        IF rtb_IP_boBMS_HV_REL_ON_BB3 THEN 
            Count_k := REAL_TO_LREAL(rtb_Add_m);
        ELSE 
            Count_k := 65535.0;
        END_IF;

        (* End of Switch: '<S128>/Switch2' *)
        (* End of Outputs for SubSystem: '<S676>/BatteryPackSignals' *)
        

        (* Switch: '<S128>/Switch3' incorporates:
         *  Constant: '<S128>/Constant5'
         *  Constant: '<S129>/Constant'
         *  Constant: '<S130>/Constant'
         *  Constant: '<S131>/Constant'
         *  Constant: '<S132>/Constant'
         *  Constant: '<S133>/Constant'
         *  Constant: '<S134>/Constant'
         *  Constant: '<S135>/Constant'
         *  Constant: '<S136>/Constant'
         *  Constant: '<S137>/Constant'
         *  Logic: '<S128>/AND'
         *  Logic: '<S128>/AND1'
         *  Logic: '<S128>/AND2'
         *  RelationalOperator: '<S129>/Compare'
         *  RelationalOperator: '<S130>/Compare'
         *  RelationalOperator: '<S131>/Compare'
         *  RelationalOperator: '<S132>/Compare'
         *  RelationalOperator: '<S133>/Compare'
         *  RelationalOperator: '<S134>/Compare'
         *  RelationalOperator: '<S135>/Compare'
         *  RelationalOperator: '<S136>/Compare'
         *  RelationalOperator: '<S137>/Compare'
         *  Switch: '<S128>/Switch4'
         *  Switch: '<S128>/Switch5' *)

        IF ((rtb_Uk1 >= 15.0) AND (rtb_UnitDelay2 >= 15.0)) AND (Count_k >= 15.0) THEN 
            rtb_Switch3 := CurrentReductionConstant_Lvl3;
        ELSIF ((rtb_Uk1 >= 10.0) AND (rtb_UnitDelay2 >= 10.0)) AND (Count_k >= 10.0) THEN 
            (* Switch: '<S128>/Switch4' incorporates:
             *  Constant: '<S128>/Constant3' *)
            rtb_Switch3 := CurrentReductionConstant_Lvl2;
        ELSIF ((rtb_Uk1 >= 5.0) AND (rtb_UnitDelay2 >= 5.0)) AND (Count_k >= 5.0) THEN 
            (* Switch: '<S128>/Switch5' incorporates:
             *  Constant: '<S128>/Constant4'
             *  Switch: '<S128>/Switch4' *)
            rtb_Switch3 := CurrentReductionConstant_Lvl1;
        ELSE 
            (* Switch: '<S128>/Switch5' incorporates:
             *  Constant: '<S128>/Constant6'
             *  Switch: '<S128>/Switch4' *)
            rtb_Switch3 := CurrentReductionConstant_Lvl0;
        END_IF;

        (* End of Switch: '<S128>/Switch3' *)
        

        (* Outputs for Atomic SubSystem: '<S676>/BatteryPackSignals' *)
        (* Product: '<S110>/Product2' incorporates:
         *  Constant: '<S110>/Constant'
         *  Constant: '<S110>/Constant5'
         *  Constant: '<S110>/Constant6'
         *  Constant: '<S126>/Constant'
         *  Logic: '<S110>/AND'
         *  MinMax: '<S110>/Min'
         *  RelationalOperator: '<S126>/Compare'
         *  RelationalOperator: '<S127>/Compare'
         *  SignalConversion: '<S682>/BusConversion_InsertedFor_IT_BatterySignal_Databus_at_inport_0'
         *  Sum: '<S110>/Add' *)

        IF rtb_NOT_m5 THEN 
            b_temp3 := MIN(rtb_Switch5_bs, rtb_Add_ci);
            temp3 := MIN(b_temp3, rtb_Divide_h) * USINT_TO_REAL(rtb_ExtractDesiredBits_bk_tmp);
        ELSE 
            temp3 := 0.0;
        END_IF;

        i0_BattChargeFcn(ssMethodType := SS_OUTPUT, MaxChargeCurr_fb := rtb_UnitDelay, MaxChargeCurrentBatt := temp3, ChargeStopPressed := rtb_IT_boChargeStop_Button, HV_ON_Batt1 := rtb_IP_boBMS_HV_REL_ON_BB1, HV_ON_Batt2 := rtb_IP_boBMS_HV_REL_ON_BB2, HV_ON_Batt3 := rtb_IP_boBMS_HV_REL_ON_BB3, Ibatt1 := rtb_Add_ki5, Ibatt2 := rtb_Add_ir, Ibatt3 := rtb_Add_m, Fcn_available := (UnexpectedBattChargingFcn_Available AND (rtb_ExtractDesiredBits_bk_tmp > 1)) AND ( NOT rtb_FL_boKL15_Disable), CurrentReductionConstant := rtb_Switch3, CurrentLB_f := CurrentLB, CurrentUB_c := CurrentUB);
        FL_sST_MaxChargeCurrent := i0_BattChargeFcn.FL_sST_MaxChargeCurrent;
        REQ_HV_Open_Batt2 := i0_BattChargeFcn.REQ_HV_Open_Batt2;
        REQ_HV_Open_Batt3 := i0_BattChargeFcn.REQ_HV_Open_Batt3;
        REQ_HV_Open_Batt1 := i0_BattChargeFcn.REQ_HV_Open_Batt1;
        BatteryReadyToShutDown := i0_BattChargeFcn.BatteryReadyToShutDown;
        (* End of Outputs for SubSystem: '<S676>/BatteryPackSignals' *)
        

        (* Switch: '<S116>/Switch' incorporates:
         *  Abs: '<S116>/Abs'
         *  Abs: '<S116>/Abs1'
         *  Abs: '<S116>/Abs2'
         *  Constant: '<S116>/Constant'
         *  Constant: '<S187>/Constant'
         *  Constant: '<S188>/Constant'
         *  Constant: '<S189>/Constant'
         *  Logic: '<S116>/AND'
         *  Logic: '<S116>/AND1'
         *  Logic: '<S116>/AND2'
         *  RelationalOperator: '<S187>/Compare'
         *  RelationalOperator: '<S188>/Compare'
         *  RelationalOperator: '<S189>/Compare'
         *  SignalConversion: '<S682>/BusConversion_InsertedFor_IT_BatterySignal_Databus_at_inport_0' *)

        IF UnexpectedBattChargingFcn_Available THEN 
            (* Outputs for Atomic SubSystem: '<S676>/BatteryPackSignals' *)
            rtb_IT_boChargeStop_Button := ((((ABS(rtb_Add_ki5) <= 1.0) AND (ABS(rtb_Add_ir) <= 1.0)) AND (ABS(rtb_Add_m) <= 1.0)) AND rtb_IT_boUDC_SafeToShutdown) OR (rtb_IT_boUDC_SafeToShutdown AND BatteryReadyToShutDown);
            (* End of Outputs for SubSystem: '<S676>/BatteryPackSignals' *)
        ELSE 
            rtb_IT_boChargeStop_Button := rtb_IT_boUDC_SafeToShutdown;
        END_IF;

        (* End of Switch: '<S116>/Switch' *)
        

        (* SignalConversion: '<S13>/TmpSignal ConversionAtChart_REQ_MAIN_MINUSInport4' *)
        i0_Chart_REQ_MAIN_MINUS(ssMethodType := SS_OUTPUT, In := rtb_Out_bl, CM_SafeToSD := rtb_IT_boChargeStop_Button, KL15_CM_disable := rtb_FL_boKL15_Disable, System_ESD := rtb_UnitDelay1_d, System_SD := rtb_UnitDelay1_d, b_Reset := rtb_FL_boSS_BDU_Reset);
        REQ_MainHV_ON_MINUS_g := i0_Chart_REQ_MAIN_MINUS.REQ_MainHV_ON_MINUS;
        (* Logic: '<S21>/AND3' incorporates:
         *  Constant: '<S13>/Constant'
         *  RelationalOperator: '<S29>/FixPt Relational Operator'
         *  UnitDelay: '<S29>/Delay Input1'
         *
         * Block description for '<S29>/Delay Input1':
         *  
         *  Store in Global RAM *)
        rtb_IT_boChargeStop_Button := (DelayInput1_DSTATE > 0.0) AND rtb_FL_boKL15_Disable;
        (* MinMax: '<S120>/Min' *)
        i0_Chart_WeldingDetection(ssMethodType := SS_OUTPUT, LoadVtg := DINT_TO_REAL(rtb_Add_kr), SystemVtg := maxV, In := rtb_IT_boChargeStop_Button);
        MainHV_Minus_Welded := i0_Chart_WeldingDetection.MainHV_Minus_Welded;
        MainHV_Plus_Welded := i0_Chart_WeldingDetection.MainHV_Plus_Welded;
        REQ_MainHV_ON_MINUS := i0_Chart_WeldingDetection.REQ_MainHV_ON_MINUS;
        REQ_MainHV_ON_PLUS := i0_Chart_WeldingDetection.REQ_MainHV_ON_PLUS;
        WeldingDetection_Status := i0_Chart_WeldingDetection.WeldingDetection_Status;
        (* UnitDelay: '<S21>/Unit Delay' *)
        rtb_System_SD_ErrorCode := UnitDelay_DSTATE_i;
        (* Chart: '<S21>/Chart4' *)
        (* Gateway: ChiefMaster/Flow Logic/BDU Control/BDUSystem/Subsystem1/Chart4 *)
        (* During: ChiefMaster/Flow Logic/BDU Control/BDUSystem/Subsystem1/Chart4 *)
        temp1 := FALSE;
        temp2 := FALSE;

        IF is_active_c46_ChiefMaster = 0 THEN 
            (* Entry: ChiefMaster/Flow Logic/BDU Control/BDUSystem/Subsystem1/Chart4 *)
            is_active_c46_ChiefMaster := 1;
            (* Entry Internal: ChiefMaster/Flow Logic/BDU Control/BDUSystem/Subsystem1/Chart4 *)
            (* Transition: '<S28>:2' *)
            is_c46_ChiefMaster := ChiefMaster_IN_Default_e2;
            (* Entry 'Default': '<S28>:1' *)
            (* '<S28>:1:2' Out = false *)
            rtb_Out_k := FALSE;
            temp1 := TRUE;
        ELSE 

            CASE is_c46_ChiefMaster OF
                ChiefMaster_IN_Default_e2: 
                    (* During 'Default': '<S28>:1' *)
                    (* '<S28>:5:1' sf_internal_predicateOutput = In == true; *)

                    IF rtb_IT_boChargeStop_Button THEN 
                        (* Transition: '<S28>:5' *)
                        is_c46_ChiefMaster := ChiefMaster_IN_Default1;
                        (* Entry 'Default1': '<S28>:4' *)
                        (* '<S28>:4:2' Out = true *)
                        rtb_Out_k := TRUE;
                        temp2 := TRUE;
                    ELSE 
                        (* '<S28>:1:2' Out = false *)
                        rtb_Out_k := FALSE;
                        temp1 := TRUE;
                    END_IF;

                ELSE
                    (* During 'Default1': '<S28>:4' *)
                    (* '<S28>:9:1' sf_internal_predicateOutput = WeldingDetection_Status == 1 ||... *)
                    (* '<S28>:9:2' WeldingDetection_Status == 2; *)

                    IF (rtb_System_SD_ErrorCode = 1) OR (rtb_System_SD_ErrorCode = 2) THEN 
                        (* Transition: '<S28>:9' *)
                        is_c46_ChiefMaster := ChiefMaster_IN_Default_e2;
                        (* Entry 'Default': '<S28>:1' *)
                        (* '<S28>:1:2' Out = false *)
                        rtb_Out_k := FALSE;
                        temp1 := TRUE;
                    ELSE 
                        (* '<S28>:4:2' Out = true *)
                        rtb_Out_k := TRUE;
                        temp2 := TRUE;
                    END_IF;

            END_CASE;

        END_IF;


        IF temp2 THEN 
            (* Switch: '<S13>/Switch' *)
            DO_REQ_MainHV_ON_MINUS := REQ_MainHV_ON_MINUS;
            (* Switch: '<S13>/Switch1' *)
            DO_REQ_MainHV_ON_PLUS := REQ_MainHV_ON_PLUS;
        END_IF;


        IF temp1 THEN 
            (* Switch: '<S13>/Switch' *)
            DO_REQ_MainHV_ON_MINUS := REQ_MainHV_ON_MINUS_g;
            (* Switch: '<S13>/Switch1' incorporates:
             *  Constant: '<S18>/Constant'
             *  Logic: '<S13>/AND5'
             *  RelationalOperator: '<S18>/Compare'
             *  RelationalOperator: '<S19>/Compare' *)
            DO_REQ_MainHV_ON_PLUS := ((Precharge_Satus = 1.0) AND rtb_IT_boHW_MainHV_Minus_FB) AND REQ_MainHV_ON_MINUS_g;
        END_IF;

        (* End of Chart: '<S21>/Chart4' *)
        

        (* Chart: '<S20>/Chart_Main_Minus_Status' incorporates:
         *  Constant: '<S20>/Constant2' *)
        (* Gateway: ChiefMaster/Flow Logic/BDU Control/BDUSystem/Subsystem/Chart_Main_Minus_Status *)
        (* During: ChiefMaster/Flow Logic/BDU Control/BDUSystem/Subsystem/Chart_Main_Minus_Status *)

        IF is_active_c40_ChiefMaster = 0 THEN 
            (* Entry: ChiefMaster/Flow Logic/BDU Control/BDUSystem/Subsystem/Chart_Main_Minus_Status *)
            is_active_c40_ChiefMaster := 1;
            (* Entry Internal: ChiefMaster/Flow Logic/BDU Control/BDUSystem/Subsystem/Chart_Main_Minus_Status *)
            (* Transition: '<S26>:2' *)
            is_c40_ChiefMaster := ChiefMaster_IN_Default_e2;
            (* Entry 'Default': '<S26>:1' *)
            (* '<S26>:1:2' MainHV_Minus_Status = 0 *)
            MainHV_Minus_Status := 0.0;
        ELSE 

            CASE is_c40_ChiefMaster OF
                ChiefMaster_IN_Default_e2: 
                    (* During 'Default': '<S26>:1' *)
                    (* '<S26>:10:1' sf_internal_predicateOutput = REQ_MainHV_ON_MINUS == false &&... *)
                    (* '<S26>:10:2' CMShutdown == false; *)

                    IF ( NOT DO_REQ_MainHV_ON_MINUS) AND ( NOT rtb_FL_boCMSleep) THEN 
                        (* Transition: '<S26>:10' *)
                        is_c40_ChiefMaster := ChiefMaster_IN_hold_a;
                        temporalCounter_i1_k(timerAction := 1, maxTime := 0);
                        (* Entry 'hold': '<S26>:9' *)
                        (* '<S26>:9:2' MainHV_Minus_Status = 0 *)
                        MainHV_Minus_Status := 0.0;
                    ELSE 
                        (* '<S26>:1:2' MainHV_Minus_Status = 0 *)
                        MainHV_Minus_Status := 0.0;
                    END_IF;

                ChiefMaster_IN_Error_p: 
                    (* During 'Error': '<S26>:16' *)
                    (* '<S26>:51:1' sf_internal_predicateOutput = CMShutdown == true; *)

                    IF rtb_FL_boCMSleep THEN 
                        (* Transition: '<S26>:51' *)
                        is_c40_ChiefMaster := ChiefMaster_IN_Default_e2;
                        (* Entry 'Default': '<S26>:1' *)
                        (* '<S26>:1:2' MainHV_Minus_Status = 0 *)
                        MainHV_Minus_Status := 0.0;
                    ELSE 
                        (* '<S26>:16:2' MainHV_Minus_Status = 3 *)
                        MainHV_Minus_Status := 3.0;
                    END_IF;

                ChiefMaster_IN_closed: 
                    (* During 'closed': '<S26>:38' *)
                    (* '<S26>:44:1' sf_internal_predicateOutput = REQ_MainHV_ON_MINUS == false; *)

                    IF  NOT DO_REQ_MainHV_ON_MINUS THEN 
                        (* Transition: '<S26>:44' *)
                        (* Transition: '<S26>:45' *)
                        (* Transition: '<S26>:49' *)
                        is_c40_ChiefMaster := ChiefMaster_IN_hold_a;
                        temporalCounter_i1_k(timerAction := 1, maxTime := 0);
                        (* Entry 'hold': '<S26>:9' *)
                        (* '<S26>:9:2' MainHV_Minus_Status = 0 *)
                        MainHV_Minus_Status := 0.0;
                    ELSE 
                        (* '<S26>:41:1' sf_internal_predicateOutput = MainHV_ON_Minus_FB == false; *)

                        IF  NOT rtb_IT_boHW_MainHV_Minus_FB THEN 
                            (* Transition: '<S26>:41' *)
                            (* Transition: '<S26>:42' *)
                            (* Transition: '<S26>:29' *)
                            (* Transition: '<S26>:27' *)
                            is_c40_ChiefMaster := ChiefMaster_IN_Error_p;
                            (* Entry 'Error': '<S26>:16' *)
                            (* '<S26>:16:2' MainHV_Minus_Status = 3 *)
                            MainHV_Minus_Status := 3.0;
                        ELSE 
                            (* '<S26>:38:2' MainHV_Minus_Status = 2 *)
                            MainHV_Minus_Status := 2.0;
                        END_IF;

                    END_IF;

                ChiefMaster_IN_hold_a: 
                    (* During 'hold': '<S26>:9' *)
                    (* '<S26>:5:1' sf_internal_predicateOutput = MainHV_ON_Minus_FB == false; *)

                    IF  NOT rtb_IT_boHW_MainHV_Minus_FB THEN 
                        (* Transition: '<S26>:5' *)
                        is_c40_ChiefMaster := ChiefMaster_IN_open;
                        (* Entry 'open': '<S26>:4' *)
                        (* '<S26>:4:2' MainHV_Minus_Status = 1 *)
                        MainHV_Minus_Status := 1.0;
                    ELSE 
                        (* '<S26>:17:1' sf_internal_predicateOutput = after(DelayTime_s,sec); *)
                        temporalCounter_i1_k(timerAction := 2, maxTime := TRUNC(REAL_TO_LREAL(MainHV_StatusDelay) * 1000.0));

                        IF temporalCounter_i1_k.done THEN 
                            (* Transition: '<S26>:17' *)
                            is_c40_ChiefMaster := ChiefMaster_IN_Error_p;
                            (* Entry 'Error': '<S26>:16' *)
                            (* '<S26>:16:2' MainHV_Minus_Status = 3 *)
                            MainHV_Minus_Status := 3.0;
                        ELSE 
                            (* '<S26>:9:2' MainHV_Minus_Status = 0 *)
                            MainHV_Minus_Status := 0.0;
                        END_IF;

                    END_IF;

                ChiefMaster_IN_hold1: 
                    (* During 'hold1': '<S26>:23' *)
                    (* '<S26>:39:1' sf_internal_predicateOutput = MainHV_ON_Minus_FB == true; *)

                    IF rtb_IT_boHW_MainHV_Minus_FB THEN 
                        (* Transition: '<S26>:39' *)
                        is_c40_ChiefMaster := ChiefMaster_IN_closed;
                        (* Entry 'closed': '<S26>:38' *)
                        (* '<S26>:38:2' MainHV_Minus_Status = 2 *)
                        MainHV_Minus_Status := 2.0;
                    ELSE 
                        (* '<S26>:26:1' sf_internal_predicateOutput = after(DelayTime_s,sec); *)
                        temporalCounter_i1_k(timerAction := 2, maxTime := TRUNC(REAL_TO_LREAL(MainHV_StatusDelay) * 1000.0));

                        IF temporalCounter_i1_k.done THEN 
                            (* Transition: '<S26>:26' *)
                            (* Transition: '<S26>:29' *)
                            (* Transition: '<S26>:27' *)
                            is_c40_ChiefMaster := ChiefMaster_IN_Error_p;
                            (* Entry 'Error': '<S26>:16' *)
                            (* '<S26>:16:2' MainHV_Minus_Status = 3 *)
                            MainHV_Minus_Status := 3.0;
                        ELSE 
                            (* '<S26>:23:2' MainHV_Minus_Status = 1 *)
                            MainHV_Minus_Status := 1.0;
                        END_IF;

                    END_IF;

                ELSE
                    (* During 'open': '<S26>:4' *)
                    (* '<S26>:11:1' sf_internal_predicateOutput = REQ_MainHV_ON_MINUS == true; *)

                    IF DO_REQ_MainHV_ON_MINUS THEN 
                        (* Transition: '<S26>:11' *)
                        is_c40_ChiefMaster := ChiefMaster_IN_hold1;
                        temporalCounter_i1_k(timerAction := 1, maxTime := 0);
                        (* Entry 'hold1': '<S26>:23' *)
                        (* '<S26>:23:2' MainHV_Minus_Status = 1 *)
                        MainHV_Minus_Status := 1.0;
                    ELSE 
                        (* '<S26>:19:1' sf_internal_predicateOutput = MainHV_ON_Minus_FB == true; *)

                        IF rtb_IT_boHW_MainHV_Minus_FB THEN 
                            (* Transition: '<S26>:19' *)
                            (* Transition: '<S26>:27' *)
                            is_c40_ChiefMaster := ChiefMaster_IN_Error_p;
                            (* Entry 'Error': '<S26>:16' *)
                            (* '<S26>:16:2' MainHV_Minus_Status = 3 *)
                            MainHV_Minus_Status := 3.0;
                        ELSE 
                            (* '<S26>:4:2' MainHV_Minus_Status = 1 *)
                            MainHV_Minus_Status := 1.0;
                        END_IF;

                    END_IF;

            END_CASE;

        END_IF;

        (* End of Chart: '<S20>/Chart_Main_Minus_Status' *)
        (* End of Outputs for SubSystem: '<Root>/ChiefMaster' *)
        

        (* Constant: '<S390>/Constant4' incorporates:
         *  Constant: '<S390>/Constant'
         *  Constant: '<S390>/Constant1'
         *  Constant: '<S390>/Constant2'
         *  Constant: '<S390>/Constant3' *)
        i2_Chart_Hysteresis_LowActive(ssMethodType := SS_OUTPUT, sSignal := AI_MainHV_Plus_FB, boInitial_Value := FALSE, boValue_Activated := TRUE, boValue_Deactivated := FALSE, sLB := 5000.0, b_sUB := 10000.0);
        boOutput_o := i2_Chart_Hysteresis_LowActive.boOutput;
        (* Outputs for Atomic SubSystem: '<Root>/ChiefMaster' *)
        (* SignalConversion: '<S677>/Signal Copy4' *)
        rtb_IT_boHW_MainHV_Plus_FB := boOutput_o;
        (* Chart: '<S20>/Chart_Main_Plus_Status' incorporates:
         *  Constant: '<S20>/Constant2'
         *  SignalConversion: '<S677>/Signal Copy4' *)
        (* Gateway: ChiefMaster/Flow Logic/BDU Control/BDUSystem/Subsystem/Chart_Main_Plus_Status *)
        (* During: ChiefMaster/Flow Logic/BDU Control/BDUSystem/Subsystem/Chart_Main_Plus_Status *)

        IF is_active_c41_ChiefMaster = 0 THEN 
            (* Entry: ChiefMaster/Flow Logic/BDU Control/BDUSystem/Subsystem/Chart_Main_Plus_Status *)
            is_active_c41_ChiefMaster := 1;
            (* Entry Internal: ChiefMaster/Flow Logic/BDU Control/BDUSystem/Subsystem/Chart_Main_Plus_Status *)
            (* Transition: '<S27>:2' *)
            is_c41_ChiefMaster := ChiefMaster_IN_Default_e2;
            (* Entry 'Default': '<S27>:1' *)
            (* '<S27>:1:2' MainHV_Plus_Status = 0 *)
            MainHV_Plus_Status := 0.0;
        ELSE 

            CASE is_c41_ChiefMaster OF
                ChiefMaster_IN_Default_e2: 
                    (* During 'Default': '<S27>:1' *)
                    (* '<S27>:10:1' sf_internal_predicateOutput = REQ_MainHV_ON_PLUS == false &&... *)
                    (* '<S27>:10:2' CMShutdown == false; *)

                    IF ( NOT DO_REQ_MainHV_ON_PLUS) AND ( NOT rtb_FL_boCMSleep) THEN 
                        (* Transition: '<S27>:10' *)
                        is_c41_ChiefMaster := ChiefMaster_IN_hold_a;
                        temporalCounter_i1_he(timerAction := 1, maxTime := 0);
                        (* Entry 'hold': '<S27>:9' *)
                        (* '<S27>:9:2' MainHV_Plus_Status = 0 *)
                        MainHV_Plus_Status := 0.0;
                    ELSE 
                        (* '<S27>:1:2' MainHV_Plus_Status = 0 *)
                        MainHV_Plus_Status := 0.0;
                    END_IF;

                ChiefMaster_IN_Error_p: 
                    (* During 'Error': '<S27>:16' *)
                    (* '<S27>:50:1' sf_internal_predicateOutput = CMShutdown == true; *)

                    IF rtb_FL_boCMSleep THEN 
                        (* Transition: '<S27>:50' *)
                        is_c41_ChiefMaster := ChiefMaster_IN_Default_e2;
                        (* Entry 'Default': '<S27>:1' *)
                        (* '<S27>:1:2' MainHV_Plus_Status = 0 *)
                        MainHV_Plus_Status := 0.0;
                    ELSE 
                        (* '<S27>:16:2' MainHV_Plus_Status = 3 *)
                        MainHV_Plus_Status := 3.0;
                    END_IF;

                ChiefMaster_IN_closed: 
                    (* During 'closed': '<S27>:38' *)
                    (* '<S27>:44:1' sf_internal_predicateOutput = REQ_MainHV_ON_PLUS == false; *)

                    IF  NOT DO_REQ_MainHV_ON_PLUS THEN 
                        (* Transition: '<S27>:44' *)
                        (* Transition: '<S27>:45' *)
                        (* Transition: '<S27>:49' *)
                        is_c41_ChiefMaster := ChiefMaster_IN_hold_a;
                        temporalCounter_i1_he(timerAction := 1, maxTime := 0);
                        (* Entry 'hold': '<S27>:9' *)
                        (* '<S27>:9:2' MainHV_Plus_Status = 0 *)
                        MainHV_Plus_Status := 0.0;
                    ELSE 
                        (* '<S27>:54:1' sf_internal_predicateOutput = MainHV_ON_Plus_FB == false; *)

                        IF  NOT boOutput_o THEN 
                            (* Transition: '<S27>:54' *)
                            (* Transition: '<S27>:42' *)
                            (* Transition: '<S27>:67' *)
                            (* Transition: '<S27>:59' *)
                            is_c41_ChiefMaster := ChiefMaster_IN_Error_p;
                            (* Entry 'Error': '<S27>:16' *)
                            (* '<S27>:16:2' MainHV_Plus_Status = 3 *)
                            MainHV_Plus_Status := 3.0;
                        ELSE 
                            (* '<S27>:38:2' MainHV_Plus_Status = 2 *)
                            MainHV_Plus_Status := 2.0;
                        END_IF;

                    END_IF;

                ChiefMaster_IN_hold_a: 
                    (* During 'hold': '<S27>:9' *)
                    (* '<S27>:5:1' sf_internal_predicateOutput = MainHV_ON_Plus_FB == false; *)

                    IF  NOT boOutput_o THEN 
                        (* Transition: '<S27>:5' *)
                        is_c41_ChiefMaster := ChiefMaster_IN_open;
                        (* Entry 'open': '<S27>:4' *)
                        (* '<S27>:4:2' MainHV_Plus_Status = 1 *)
                        MainHV_Plus_Status := 1.0;
                    ELSE 
                        (* '<S27>:17:1' sf_internal_predicateOutput = after(DelayTime_s,sec); *)
                        temporalCounter_i1_he(timerAction := 2, maxTime := TRUNC(REAL_TO_LREAL(MainHV_StatusDelay) * 1000.0));

                        IF temporalCounter_i1_he.done THEN 
                            (* Transition: '<S27>:17' *)
                            is_c41_ChiefMaster := ChiefMaster_IN_Error_p;
                            (* Entry 'Error': '<S27>:16' *)
                            (* '<S27>:16:2' MainHV_Plus_Status = 3 *)
                            MainHV_Plus_Status := 3.0;
                        ELSE 
                            (* '<S27>:9:2' MainHV_Plus_Status = 0 *)
                            MainHV_Plus_Status := 0.0;
                        END_IF;

                    END_IF;

                ChiefMaster_IN_hold1: 
                    (* During 'hold1': '<S27>:23' *)
                    (* '<S27>:39:1' sf_internal_predicateOutput = MainHV_ON_Plus_FB == true; *)

                    IF boOutput_o THEN 
                        (* Transition: '<S27>:39' *)
                        is_c41_ChiefMaster := ChiefMaster_IN_closed;
                        (* Entry 'closed': '<S27>:38' *)
                        (* '<S27>:38:2' MainHV_Plus_Status = 2 *)
                        MainHV_Plus_Status := 2.0;
                    ELSE 
                        (* '<S27>:26:1' sf_internal_predicateOutput = after(DelayTime_s,sec); *)
                        temporalCounter_i1_he(timerAction := 2, maxTime := TRUNC(REAL_TO_LREAL(MainHV_StatusDelay) * 1000.0));

                        IF temporalCounter_i1_he.done THEN 
                            (* Transition: '<S27>:26' *)
                            (* Transition: '<S27>:67' *)
                            (* Transition: '<S27>:59' *)
                            is_c41_ChiefMaster := ChiefMaster_IN_Error_p;
                            (* Entry 'Error': '<S27>:16' *)
                            (* '<S27>:16:2' MainHV_Plus_Status = 3 *)
                            MainHV_Plus_Status := 3.0;
                        ELSE 
                            (* '<S27>:23:2' MainHV_Plus_Status = 1 *)
                            MainHV_Plus_Status := 1.0;
                        END_IF;

                    END_IF;

                ELSE
                    (* During 'open': '<S27>:4' *)
                    (* '<S27>:11:1' sf_internal_predicateOutput = REQ_MainHV_ON_PLUS == true; *)

                    IF DO_REQ_MainHV_ON_PLUS THEN 
                        (* Transition: '<S27>:11' *)
                        is_c41_ChiefMaster := ChiefMaster_IN_hold1;
                        temporalCounter_i1_he(timerAction := 1, maxTime := 0);
                        (* Entry 'hold1': '<S27>:23' *)
                        (* '<S27>:23:2' MainHV_Plus_Status = 1 *)
                        MainHV_Plus_Status := 1.0;
                    ELSE 
                        (* '<S27>:58:1' sf_internal_predicateOutput = MainHV_ON_Plus_FB == true; *)

                        IF boOutput_o THEN 
                            (* Transition: '<S27>:58' *)
                            (* Transition: '<S27>:59' *)
                            is_c41_ChiefMaster := ChiefMaster_IN_Error_p;
                            (* Entry 'Error': '<S27>:16' *)
                            (* '<S27>:16:2' MainHV_Plus_Status = 3 *)
                            MainHV_Plus_Status := 3.0;
                        ELSE 
                            (* '<S27>:4:2' MainHV_Plus_Status = 1 *)
                            MainHV_Plus_Status := 1.0;
                        END_IF;

                    END_IF;

            END_CASE;

        END_IF;

        (* End of Chart: '<S20>/Chart_Main_Plus_Status' *)
        (* End of Outputs for SubSystem: '<Root>/ChiefMaster' *)
        

        (* Constant: '<S389>/Constant4' incorporates:
         *  Constant: '<S389>/Constant'
         *  Constant: '<S389>/Constant1'
         *  Constant: '<S389>/Constant2'
         *  Constant: '<S389>/Constant3' *)
        i1_Chart_Hysteresis_LowActive(ssMethodType := SS_OUTPUT, sSignal := AI_DCHV_Minus_FB, boInitial_Value := FALSE, boValue_Activated := TRUE, boValue_Deactivated := FALSE, sLB := 5000.0, b_sUB := 10000.0);
        boOutput_a := i1_Chart_Hysteresis_LowActive.boOutput;
        (* Outputs for Atomic SubSystem: '<Root>/ChiefMaster' *)
        (* SignalConversion: '<S677>/Signal Copy13' *)
        rtb_IT_boHW_DCHV_Minus_FB := boOutput_a;
        (* Chart: '<S23>/Chart_DCMinus_Status' incorporates:
         *  Constant: '<S23>/Constant2'
         *  SignalConversion: '<S677>/Signal Copy13' *)
        (* Gateway: ChiefMaster/Flow Logic/BDU Control/BDUSystem/Subsystem3/Chart_DCMinus_Status *)
        (* During: ChiefMaster/Flow Logic/BDU Control/BDUSystem/Subsystem3/Chart_DCMinus_Status *)

        IF is_active_c53_ChiefMaster = 0 THEN 
            (* Entry: ChiefMaster/Flow Logic/BDU Control/BDUSystem/Subsystem3/Chart_DCMinus_Status *)
            is_active_c53_ChiefMaster := 1;
            (* Entry Internal: ChiefMaster/Flow Logic/BDU Control/BDUSystem/Subsystem3/Chart_DCMinus_Status *)
            (* Transition: '<S31>:2' *)
            is_c53_ChiefMaster := ChiefMaster_IN_Default_e2;
            (* Entry 'Default': '<S31>:1' *)
            (* '<S31>:1:2' HV_Minus_Status = 0 *)
            rtb_Uk1 := 0.0;
        ELSE 

            CASE is_c53_ChiefMaster OF
                ChiefMaster_IN_Default_e2: 
                    (* During 'Default': '<S31>:1' *)
                    (* '<S31>:10:1' sf_internal_predicateOutput = REQ_HV_ON_MINUS == false &&... *)
                    (* '<S31>:10:2' CMSleep == false; *)

                    IF ( NOT DO_REQ_DC_ON_PLUS) AND ( NOT rtb_FL_boCMSleep) THEN 
                        (* Transition: '<S31>:10' *)
                        is_c53_ChiefMaster := ChiefMaster_IN_hold_a;
                        temporalCounter_i1_n(timerAction := 1, maxTime := 0);
                        (* Entry 'hold': '<S31>:9' *)
                        (* '<S31>:9:2' HV_Minus_Status = 0 *)
                        rtb_Uk1 := 0.0;
                    ELSE 
                        (* '<S31>:1:2' HV_Minus_Status = 0 *)
                        rtb_Uk1 := 0.0;
                    END_IF;

                ChiefMaster_IN_Error_p: 
                    (* During 'Error': '<S31>:16' *)
                    (* '<S31>:51:1' sf_internal_predicateOutput = CMSleep == true; *)

                    IF rtb_FL_boCMSleep THEN 
                        (* Transition: '<S31>:51' *)
                        is_c53_ChiefMaster := ChiefMaster_IN_Default_e2;
                        (* Entry 'Default': '<S31>:1' *)
                        (* '<S31>:1:2' HV_Minus_Status = 0 *)
                        rtb_Uk1 := 0.0;
                    ELSE 
                        (* '<S31>:16:2' HV_Minus_Status = 3 *)
                        rtb_Uk1 := 3.0;
                    END_IF;

                ChiefMaster_IN_closed: 
                    (* During 'closed': '<S31>:38' *)
                    (* '<S31>:44:1' sf_internal_predicateOutput = REQ_HV_ON_MINUS == false; *)

                    IF  NOT DO_REQ_DC_ON_PLUS THEN 
                        (* Transition: '<S31>:44' *)
                        (* Transition: '<S31>:45' *)
                        (* Transition: '<S31>:49' *)
                        is_c53_ChiefMaster := ChiefMaster_IN_hold_a;
                        temporalCounter_i1_n(timerAction := 1, maxTime := 0);
                        (* Entry 'hold': '<S31>:9' *)
                        (* '<S31>:9:2' HV_Minus_Status = 0 *)
                        rtb_Uk1 := 0.0;
                    ELSE 
                        (* '<S31>:41:1' sf_internal_predicateOutput = HV_ON_Minus_FB == false; *)

                        IF  NOT boOutput_a THEN 
                            (* Transition: '<S31>:41' *)
                            (* Transition: '<S31>:42' *)
                            (* Transition: '<S31>:29' *)
                            (* Transition: '<S31>:27' *)
                            is_c53_ChiefMaster := ChiefMaster_IN_Error_p;
                            (* Entry 'Error': '<S31>:16' *)
                            (* '<S31>:16:2' HV_Minus_Status = 3 *)
                            rtb_Uk1 := 3.0;
                        ELSE 
                            (* '<S31>:38:2' HV_Minus_Status = 2 *)
                            rtb_Uk1 := 2.0;
                        END_IF;

                    END_IF;

                ChiefMaster_IN_hold_a: 
                    (* During 'hold': '<S31>:9' *)
                    (* '<S31>:5:1' sf_internal_predicateOutput = HV_ON_Minus_FB == false; *)

                    IF  NOT boOutput_a THEN 
                        (* Transition: '<S31>:5' *)
                        is_c53_ChiefMaster := ChiefMaster_IN_open;
                        (* Entry 'open': '<S31>:4' *)
                        (* '<S31>:4:2' HV_Minus_Status = 1 *)
                        rtb_Uk1 := 1.0;
                    ELSE 
                        (* '<S31>:17:1' sf_internal_predicateOutput = after(DelayTime_s,sec); *)
                        temporalCounter_i1_n(timerAction := 2, maxTime := TRUNC(REAL_TO_LREAL(MainHV_StatusDelay) * 1000.0));

                        IF temporalCounter_i1_n.done THEN 
                            (* Transition: '<S31>:17' *)
                            is_c53_ChiefMaster := ChiefMaster_IN_Error_p;
                            (* Entry 'Error': '<S31>:16' *)
                            (* '<S31>:16:2' HV_Minus_Status = 3 *)
                            rtb_Uk1 := 3.0;
                        ELSE 
                            (* '<S31>:9:2' HV_Minus_Status = 0 *)
                            rtb_Uk1 := 0.0;
                        END_IF;

                    END_IF;

                ChiefMaster_IN_hold1: 
                    (* During 'hold1': '<S31>:23' *)
                    (* '<S31>:39:1' sf_internal_predicateOutput = HV_ON_Minus_FB == true; *)

                    IF boOutput_a THEN 
                        (* Transition: '<S31>:39' *)
                        is_c53_ChiefMaster := ChiefMaster_IN_closed;
                        (* Entry 'closed': '<S31>:38' *)
                        (* '<S31>:38:2' HV_Minus_Status = 2 *)
                        rtb_Uk1 := 2.0;
                    ELSE 
                        (* '<S31>:26:1' sf_internal_predicateOutput = after(DelayTime_s,sec); *)
                        temporalCounter_i1_n(timerAction := 2, maxTime := TRUNC(REAL_TO_LREAL(MainHV_StatusDelay) * 1000.0));

                        IF temporalCounter_i1_n.done THEN 
                            (* Transition: '<S31>:26' *)
                            (* Transition: '<S31>:29' *)
                            (* Transition: '<S31>:27' *)
                            is_c53_ChiefMaster := ChiefMaster_IN_Error_p;
                            (* Entry 'Error': '<S31>:16' *)
                            (* '<S31>:16:2' HV_Minus_Status = 3 *)
                            rtb_Uk1 := 3.0;
                        ELSE 
                            (* '<S31>:23:2' HV_Minus_Status = 1 *)
                            rtb_Uk1 := 1.0;
                        END_IF;

                    END_IF;

                ELSE
                    (* During 'open': '<S31>:4' *)
                    (* '<S31>:11:1' sf_internal_predicateOutput = REQ_HV_ON_MINUS == true; *)

                    IF DO_REQ_DC_ON_PLUS THEN 
                        (* Transition: '<S31>:11' *)
                        is_c53_ChiefMaster := ChiefMaster_IN_hold1;
                        temporalCounter_i1_n(timerAction := 1, maxTime := 0);
                        (* Entry 'hold1': '<S31>:23' *)
                        (* '<S31>:23:2' HV_Minus_Status = 1 *)
                        rtb_Uk1 := 1.0;
                    ELSE 
                        (* '<S31>:19:1' sf_internal_predicateOutput = HV_ON_Minus_FB == true; *)

                        IF boOutput_a THEN 
                            (* Transition: '<S31>:19' *)
                            (* Transition: '<S31>:27' *)
                            is_c53_ChiefMaster := ChiefMaster_IN_Error_p;
                            (* Entry 'Error': '<S31>:16' *)
                            (* '<S31>:16:2' HV_Minus_Status = 3 *)
                            rtb_Uk1 := 3.0;
                        ELSE 
                            (* '<S31>:4:2' HV_Minus_Status = 1 *)
                            rtb_Uk1 := 1.0;
                        END_IF;

                    END_IF;

            END_CASE;

        END_IF;

        (* End of Chart: '<S23>/Chart_DCMinus_Status' *)
        (* End of Outputs for SubSystem: '<Root>/ChiefMaster' *)
        

        (* Constant: '<S391>/Constant4' incorporates:
         *  Constant: '<S391>/Constant'
         *  Constant: '<S391>/Constant1'
         *  Constant: '<S391>/Constant2'
         *  Constant: '<S391>/Constant3' *)
        i3_Chart_Hysteresis_LowActive(ssMethodType := SS_OUTPUT, sSignal := AI_DCHV_Plus_FB, boInitial_Value := FALSE, boValue_Activated := TRUE, boValue_Deactivated := FALSE, sLB := 5000.0, b_sUB := 10000.0);
        boOutput := i3_Chart_Hysteresis_LowActive.boOutput;
        (* Outputs for Atomic SubSystem: '<Root>/ChiefMaster' *)
        (* SignalConversion: '<S677>/Signal Copy12' *)
        rtb_IT_boHW_DCHV_Plus_FB := boOutput;
        (* Chart: '<S23>/Chart_DCPlus_Status' incorporates:
         *  Constant: '<S23>/Constant2'
         *  SignalConversion: '<S677>/Signal Copy12' *)
        (* Gateway: ChiefMaster/Flow Logic/BDU Control/BDUSystem/Subsystem3/Chart_DCPlus_Status *)
        (* During: ChiefMaster/Flow Logic/BDU Control/BDUSystem/Subsystem3/Chart_DCPlus_Status *)

        IF is_active_c54_ChiefMaster = 0 THEN 
            (* Entry: ChiefMaster/Flow Logic/BDU Control/BDUSystem/Subsystem3/Chart_DCPlus_Status *)
            is_active_c54_ChiefMaster := 1;
            (* Entry Internal: ChiefMaster/Flow Logic/BDU Control/BDUSystem/Subsystem3/Chart_DCPlus_Status *)
            (* Transition: '<S32>:2' *)
            is_c54_ChiefMaster := ChiefMaster_IN_Default_e2;
            (* Entry 'Default': '<S32>:1' *)
            (* '<S32>:1:2' HV_Plus_Status = 0 *)
            rtb_UnitDelay2 := 0.0;
        ELSE 

            CASE is_c54_ChiefMaster OF
                ChiefMaster_IN_Default_e2: 
                    (* During 'Default': '<S32>:1' *)
                    (* '<S32>:10:1' sf_internal_predicateOutput = REQ_HV_ON_PLUS == false &&... *)
                    (* '<S32>:10:2' CMSleep == false; *)

                    IF ( NOT DO_REQ_DC_ON_PLUS) AND ( NOT rtb_FL_boCMSleep) THEN 
                        (* Transition: '<S32>:10' *)
                        is_c54_ChiefMaster := ChiefMaster_IN_hold_a;
                        temporalCounter_i1_a(timerAction := 1, maxTime := 0);
                        (* Entry 'hold': '<S32>:9' *)
                        (* '<S32>:9:2' HV_Plus_Status = 0 *)
                        rtb_UnitDelay2 := 0.0;
                    ELSE 
                        (* '<S32>:1:2' HV_Plus_Status = 0 *)
                        rtb_UnitDelay2 := 0.0;
                    END_IF;

                ChiefMaster_IN_Error_p: 
                    (* During 'Error': '<S32>:16' *)
                    (* '<S32>:51:1' sf_internal_predicateOutput = CMSleep == true; *)

                    IF rtb_FL_boCMSleep THEN 
                        (* Transition: '<S32>:51' *)
                        is_c54_ChiefMaster := ChiefMaster_IN_Default_e2;
                        (* Entry 'Default': '<S32>:1' *)
                        (* '<S32>:1:2' HV_Plus_Status = 0 *)
                        rtb_UnitDelay2 := 0.0;
                    ELSE 
                        (* '<S32>:16:2' HV_Plus_Status = 3 *)
                        rtb_UnitDelay2 := 3.0;
                    END_IF;

                ChiefMaster_IN_closed: 
                    (* During 'closed': '<S32>:38' *)
                    (* '<S32>:44:1' sf_internal_predicateOutput = REQ_HV_ON_PLUS == false; *)

                    IF  NOT DO_REQ_DC_ON_PLUS THEN 
                        (* Transition: '<S32>:44' *)
                        (* Transition: '<S32>:45' *)
                        (* Transition: '<S32>:49' *)
                        is_c54_ChiefMaster := ChiefMaster_IN_hold_a;
                        temporalCounter_i1_a(timerAction := 1, maxTime := 0);
                        (* Entry 'hold': '<S32>:9' *)
                        (* '<S32>:9:2' HV_Plus_Status = 0 *)
                        rtb_UnitDelay2 := 0.0;
                    ELSE 
                        (* '<S32>:41:1' sf_internal_predicateOutput = HV_ON_Plus_FB == false; *)

                        IF  NOT boOutput THEN 
                            (* Transition: '<S32>:41' *)
                            (* Transition: '<S32>:42' *)
                            (* Transition: '<S32>:29' *)
                            (* Transition: '<S32>:27' *)
                            is_c54_ChiefMaster := ChiefMaster_IN_Error_p;
                            (* Entry 'Error': '<S32>:16' *)
                            (* '<S32>:16:2' HV_Plus_Status = 3 *)
                            rtb_UnitDelay2 := 3.0;
                        ELSE 
                            (* '<S32>:38:2' HV_Plus_Status = 2 *)
                            rtb_UnitDelay2 := 2.0;
                        END_IF;

                    END_IF;

                ChiefMaster_IN_hold_a: 
                    (* During 'hold': '<S32>:9' *)
                    (* '<S32>:5:1' sf_internal_predicateOutput = HV_ON_Plus_FB == false; *)

                    IF  NOT boOutput THEN 
                        (* Transition: '<S32>:5' *)
                        is_c54_ChiefMaster := ChiefMaster_IN_open;
                        (* Entry 'open': '<S32>:4' *)
                        (* '<S32>:4:2' HV_Plus_Status = 1 *)
                        rtb_UnitDelay2 := 1.0;
                    ELSE 
                        (* '<S32>:17:1' sf_internal_predicateOutput = after(DelayTime_s,sec); *)
                        temporalCounter_i1_a(timerAction := 2, maxTime := TRUNC(REAL_TO_LREAL(MainHV_StatusDelay) * 1000.0));

                        IF temporalCounter_i1_a.done THEN 
                            (* Transition: '<S32>:17' *)
                            is_c54_ChiefMaster := ChiefMaster_IN_Error_p;
                            (* Entry 'Error': '<S32>:16' *)
                            (* '<S32>:16:2' HV_Plus_Status = 3 *)
                            rtb_UnitDelay2 := 3.0;
                        ELSE 
                            (* '<S32>:9:2' HV_Plus_Status = 0 *)
                            rtb_UnitDelay2 := 0.0;
                        END_IF;

                    END_IF;

                ChiefMaster_IN_hold1: 
                    (* During 'hold1': '<S32>:23' *)
                    (* '<S32>:39:1' sf_internal_predicateOutput = HV_ON_Plus_FB == true; *)

                    IF boOutput THEN 
                        (* Transition: '<S32>:39' *)
                        is_c54_ChiefMaster := ChiefMaster_IN_closed;
                        (* Entry 'closed': '<S32>:38' *)
                        (* '<S32>:38:2' HV_Plus_Status = 2 *)
                        rtb_UnitDelay2 := 2.0;
                    ELSE 
                        (* '<S32>:26:1' sf_internal_predicateOutput = after(DelayTime_s,sec); *)
                        temporalCounter_i1_a(timerAction := 2, maxTime := TRUNC(REAL_TO_LREAL(MainHV_StatusDelay) * 1000.0));

                        IF temporalCounter_i1_a.done THEN 
                            (* Transition: '<S32>:26' *)
                            (* Transition: '<S32>:29' *)
                            (* Transition: '<S32>:27' *)
                            is_c54_ChiefMaster := ChiefMaster_IN_Error_p;
                            (* Entry 'Error': '<S32>:16' *)
                            (* '<S32>:16:2' HV_Plus_Status = 3 *)
                            rtb_UnitDelay2 := 3.0;
                        ELSE 
                            (* '<S32>:23:2' HV_Plus_Status = 1 *)
                            rtb_UnitDelay2 := 1.0;
                        END_IF;

                    END_IF;

                ELSE
                    (* During 'open': '<S32>:4' *)
                    (* '<S32>:11:1' sf_internal_predicateOutput = REQ_HV_ON_PLUS == true; *)

                    IF DO_REQ_DC_ON_PLUS THEN 
                        (* Transition: '<S32>:11' *)
                        is_c54_ChiefMaster := ChiefMaster_IN_hold1;
                        temporalCounter_i1_a(timerAction := 1, maxTime := 0);
                        (* Entry 'hold1': '<S32>:23' *)
                        (* '<S32>:23:2' HV_Plus_Status = 1 *)
                        rtb_UnitDelay2 := 1.0;
                    ELSE 
                        (* '<S32>:19:1' sf_internal_predicateOutput = HV_ON_Plus_FB == true; *)

                        IF boOutput THEN 
                            (* Transition: '<S32>:19' *)
                            (* Transition: '<S32>:27' *)
                            is_c54_ChiefMaster := ChiefMaster_IN_Error_p;
                            (* Entry 'Error': '<S32>:16' *)
                            (* '<S32>:16:2' HV_Plus_Status = 3 *)
                            rtb_UnitDelay2 := 3.0;
                        ELSE 
                            (* '<S32>:4:2' HV_Plus_Status = 1 *)
                            rtb_UnitDelay2 := 1.0;
                        END_IF;

                    END_IF;

            END_CASE;

        END_IF;

        (* End of Chart: '<S23>/Chart_DCPlus_Status' *)
        

        (* Chart: '<S13>/delay1' incorporates:
         *  Constant: '<S13>/Constant2' *)
        (* Gateway: ChiefMaster/Flow Logic/BDU Control/BDUSystem/delay1 *)
        (* During: ChiefMaster/Flow Logic/BDU Control/BDUSystem/delay1 *)

        IF is_active_c51_ChiefMaster = 0 THEN 
            (* Entry: ChiefMaster/Flow Logic/BDU Control/BDUSystem/delay1 *)
            is_active_c51_ChiefMaster := 1;
            (* Entry Internal: ChiefMaster/Flow Logic/BDU Control/BDUSystem/delay1 *)
            (* Transition: '<S25>:2' *)
            is_c51_ChiefMaster := ChiefMaster_IN_Default_i2;
            (* Entry 'Default': '<S25>:1' *)
            (* '<S25>:1:2' Out = false *)
            DO_REQ_DC_ON_MINUS := FALSE;
        ELSE 

            CASE is_c51_ChiefMaster OF
                ChiefMaster_IN_Actual_o: 
                    (* During 'Actual': '<S25>:11' *)
                    (* Transition: '<S25>:17' *)
                    (* '<S25>:14:1' sf_internal_predicateOutput = In == false; *)

                    IF  NOT DO_REQ_DC_ON_PLUS THEN 
                        (* Transition: '<S25>:14' *)
                        is_c51_ChiefMaster := ChiefMaster_IN_Default_i2;
                        (* Entry 'Default': '<S25>:1' *)
                        (* '<S25>:1:2' Out = false *)
                        DO_REQ_DC_ON_MINUS := FALSE;
                    ELSE 
                        (* '<S25>:11:2' Out = In *)
                        DO_REQ_DC_ON_MINUS := TRUE;
                    END_IF;

                ChiefMaster_IN_Default_i2: 
                    (* During 'Default': '<S25>:1' *)
                    (* '<S25>:5:1' sf_internal_predicateOutput = In == true; *)

                    IF DO_REQ_DC_ON_PLUS THEN 
                        (* Transition: '<S25>:5' *)
                        is_c51_ChiefMaster := ChiefMaster_IN_hold_oa;
                        temporalCounter_i1_h(timerAction := 1, maxTime := 0);
                        (* Entry 'hold': '<S25>:4' *)
                        (* '<S25>:4:2' Out = false *)
                        DO_REQ_DC_ON_MINUS := FALSE;
                    ELSE 
                        (* '<S25>:1:2' Out = false *)
                        DO_REQ_DC_ON_MINUS := FALSE;
                    END_IF;

                ELSE
                    (* During 'hold': '<S25>:4' *)
                    (* '<S25>:12:1' sf_internal_predicateOutput = after(DelayTime_ms,msec); *)
                    temporalCounter_i1_h(timerAction := 2, maxTime := TRUNC(DCHV_Minus_In_Delay_ms));

                    IF temporalCounter_i1_h.done THEN 
                        (* Transition: '<S25>:12' *)
                        is_c51_ChiefMaster := ChiefMaster_IN_Actual_o;
                        (* Entry 'Actual': '<S25>:11' *)
                        (* '<S25>:11:2' Out = In *)
                        DO_REQ_DC_ON_MINUS := DO_REQ_DC_ON_PLUS;
                    ELSE 
                        (* Transition: '<S25>:16' *)
                        (* '<S25>:14:1' sf_internal_predicateOutput = In == false; *)

                        IF  NOT DO_REQ_DC_ON_PLUS THEN 
                            (* Transition: '<S25>:14' *)
                            is_c51_ChiefMaster := ChiefMaster_IN_Default_i2;
                            (* Entry 'Default': '<S25>:1' *)
                            (* '<S25>:1:2' Out = false *)
                            DO_REQ_DC_ON_MINUS := FALSE;
                        ELSE 
                            (* '<S25>:4:2' Out = false *)
                            DO_REQ_DC_ON_MINUS := FALSE;
                        END_IF;

                    END_IF;

            END_CASE;

        END_IF;

        (* End of Chart: '<S13>/delay1' *)
        

        (* Outputs for Atomic SubSystem: '<S676>/BatteryPackSignals' *)
        (* SignalConversion: '<S698>/Signal Copy' incorporates:
         *  SignalConversion: '<S682>/BusConversion_InsertedFor_IT_BatterySignal_Databus_at_inport_0'
         *  SignalConversion: '<S699>/Signal Copy'
         *  SignalConversion: '<S700>/Signal Copy' *)
        i0_InsulationMonitoringReq(ssMethodType := SS_OUTPUT, IT_boUDC_KL15_D := rtb_IT_boUDC_KL15_D, IT_boUDC_KL15_C := rtb_IT_boUDC_KL15_C, IT_boBMS_HV_ON_BB := rtb_IT_boBMS_HV_ON_BB, IT_u8BMS_BB_No_MaxVoltage := rtb_Switch_a, IT_u8BMS_BB_No_MinVoltage := rtb_Switch2_k, IT_boBMS_SDError_BB1 := rtb_IP_boBMS_SDError_BB1, IT_boBMS_SDError_BB2 := rtb_IP_boBMS_SDError_BB2, IT_boBMS_SDError_BB3 := rtb_IP_boBMS_SDError_BB3, IT_boBMS_InsulationReadyOK_B1 := rtb_S_in, IT_boBMS_InsulationReadyOK_B2 := rtb_IP_boBatt1_Actia_Availability, IT_boBMS_InsulationReadyOK_B3 := rtb_Delay_dl, IT_boBMS_IMD_Active_BB1 := rtb_IP_boBMS_IMD_Active_BB1, IT_boBMS_IMD_Active_BB2 := rtb_IP_boBMS_IMD_Active_BB2, IT_boBMS_IMD_Active_BB3 := rtb_IP_boBMS_IMD_Active_BB3, IT_boBMS_HV_REL_ON_BB1 := rtb_IP_boBMS_HV_REL_ON_BB1, IT_boBMS_HV_REL_ON_BB2 := rtb_IP_boBMS_HV_REL_ON_BB2, IT_boBMS_HV_REL_ON_BB3 := rtb_IP_boBMS_HV_REL_ON_BB3, IT_sBMS_Batt1_Availability := DINT_TO_LREAL(rtb_IP_boBMS_Batt1_Availability), IT_sBMS_Batt2_Availability := DINT_TO_LREAL(rtb_UnitDelay5), IT_sBMS_Batt3_Availability := DINT_TO_LREAL(rtb_IP_boBMS_Batt3_Availability), IT_boUDC_EV_IsolationMeasurementRequest := rtb_IT_boUDC_EV_IsolationMeasurementRequest, FL_boSS_System_SD := System_Error, FL_boSS_System_ESD := rtb_Delay_j);
        rtb_IT_boChargeStop_Button := i0_InsulationMonitoringReq.FL_boREQ_IMD_ON_BB1;
        rtb_UnitDelay1_d := i0_InsulationMonitoringReq.FL_boREQ_IMD_ON_BB2;
        rtb_Out_bl := i0_InsulationMonitoringReq.FL_boREQ_IMD_ON_BB3;
        rtb_IMD_State_g := i0_InsulationMonitoringReq.FL_u8_IMD_State_BB1;
        rtb_System_SD_ErrorCode := i0_InsulationMonitoringReq.FL_u8_IMD_State_BB2;
        rtb_IMD_State := i0_InsulationMonitoringReq.FL_u8_IMD_State_BB3;
        (* End of Outputs for SubSystem: '<S676>/BatteryPackSignals' *)
        (* End of Outputs for SubSystem: '<Root>/ChiefMaster' *)
        

        (* Constant: '<S81>/Constant' *)
        i0_Chart_jj(ssMethodType := SS_OUTPUT, In := ContactorState_f, b_n := 5.0);
        rtb_IT_boUDC_EV_IsolationMeasurementRequest := i0_Chart_jj.Out;
        (* Outputs for Atomic SubSystem: '<Root>/ChiefMaster' *)
        (* Logic: '<S81>/AND' incorporates:
         *  Constant: '<S78>/Constant'
         *  Logic: '<S81>/AND2'
         *  RelationalOperator: '<S78>/Compare' *)
        i0_Chart1(ssMethodType := SS_OUTPUT, In := ((rtb_Switch2_k = 2.0) AND rtb_IT_boUDC_EV_IsolationMeasurementRequest) AND rtb_IT_boUDC_KL15_C);
        rtb_Out_ap := i0_Chart1.Out;
        (* End of Outputs for SubSystem: '<Root>/ChiefMaster' *)
        

        (* Constant: '<S82>/Constant' *)
        i1_Chart_jj(ssMethodType := SS_OUTPUT, In := ContactorState, b_n := 5.0);
        rtb_IT_boUDC_EV_IsolationMeasurementRequest := i1_Chart_jj.Out;
        (* Outputs for Atomic SubSystem: '<Root>/ChiefMaster' *)
        (* Logic: '<S82>/AND' incorporates:
         *  Constant: '<S79>/Constant'
         *  Logic: '<S82>/AND2'
         *  RelationalOperator: '<S79>/Compare' *)
        i1_Chart1(ssMethodType := SS_OUTPUT, In := ((rtb_Switch2_k = 3.0) AND rtb_IT_boUDC_EV_IsolationMeasurementRequest) AND rtb_IT_boUDC_KL15_C);
        rtb_Out_ap := i1_Chart1.Out;
        (* Outputs for Atomic SubSystem: '<S676>/BatteryPackSignals' *)
        (* SignalConversion: '<S698>/Signal Copy' incorporates:
         *  Outport: '<Root>/DO_KL15_BB1'
         *  RelationalOperator: '<S94>/FixPt Relational Operator'
         *  RelationalOperator: '<S95>/Compare'
         *  UnitDelay: '<S94>/Delay Input1'
         *
         * Block description for '<S94>/Delay Input1':
         *  
         *  Store in Global RAM *)
        i0_Chart_lg(ssMethodType := SS_OUTPUT, Error := rtb_IP_boBMS_SDError_BB1, KL15_reset := BOOL_TO_DINT(DO_KL15_BB1) > BOOL_TO_DINT(DelayInput1_DSTATE_g));
        rtb_IT_boUDC_EV_IsolationMeasurementRequest := i0_Chart_lg.SW_Reset;
        (* End of Outputs for SubSystem: '<S676>/BatteryPackSignals' *)
        

        (* Logic: '<S83>/NAND' *)
        i0_Chart1_l(ssMethodType := SS_OUTPUT, SW_Reset := rtb_IT_boUDC_EV_IsolationMeasurementRequest, KL_15_reset_CM := ( NOT rtb_IT_boUDC_KL15_C) AND ( NOT rtb_IT_boUDC_KL15_D));
        Count_k := i0_Chart1_l.Count;
        (* Outputs for Atomic SubSystem: '<S676>/BatteryPackSignals' *)
        (* SignalConversion: '<S699>/Signal Copy' incorporates:
         *  Outport: '<Root>/DO_KL15_BB2'
         *  RelationalOperator: '<S100>/Compare'
         *  RelationalOperator: '<S99>/FixPt Relational Operator'
         *  UnitDelay: '<S99>/Delay Input1'
         *
         * Block description for '<S99>/Delay Input1':
         *  
         *  Store in Global RAM *)
        i1_Chart_lg(ssMethodType := SS_OUTPUT, Error := rtb_IP_boBMS_SDError_BB2, KL15_reset := BOOL_TO_DINT(DO_KL15_BB2) > BOOL_TO_DINT(DelayInput1_DSTATE_n));
        rtb_IT_boUDC_EV_IsolationMeasurementRequest := i1_Chart_lg.SW_Reset;
        (* End of Outputs for SubSystem: '<S676>/BatteryPackSignals' *)
        

        (* Logic: '<S84>/NAND' *)
        i1_Chart1_l(ssMethodType := SS_OUTPUT, SW_Reset := rtb_IT_boUDC_EV_IsolationMeasurementRequest, KL_15_reset_CM := ( NOT rtb_IT_boUDC_KL15_C) AND ( NOT rtb_IT_boUDC_KL15_D));
        Count_k := i1_Chart1_l.Count;
        (* Outputs for Atomic SubSystem: '<S676>/BatteryPackSignals' *)
        (* SignalConversion: '<S700>/Signal Copy' incorporates:
         *  Outport: '<Root>/DO_KL15_BB3'
         *  RelationalOperator: '<S104>/FixPt Relational Operator'
         *  RelationalOperator: '<S105>/Compare'
         *  UnitDelay: '<S104>/Delay Input1'
         *
         * Block description for '<S104>/Delay Input1':
         *  
         *  Store in Global RAM *)
        i2_Chart_lg(ssMethodType := SS_OUTPUT, Error := rtb_IP_boBMS_SDError_BB3, KL15_reset := BOOL_TO_DINT(DO_KL15_BB3) > BOOL_TO_DINT(DelayInput1_DSTATE_e));
        rtb_IT_boUDC_EV_IsolationMeasurementRequest := i2_Chart_lg.SW_Reset;
        (* End of Outputs for SubSystem: '<S676>/BatteryPackSignals' *)
        

        (* Logic: '<S85>/NAND' *)
        i2_Chart1_l(ssMethodType := SS_OUTPUT, SW_Reset := rtb_IT_boUDC_EV_IsolationMeasurementRequest, KL_15_reset_CM := ( NOT rtb_IT_boUDC_KL15_C) AND ( NOT rtb_IT_boUDC_KL15_D));
        Count_k := i2_Chart1_l.Count;
        (* End of Outputs for SubSystem: '<Root>/ChiefMaster' *)
        

        (* Constant: '<S86>/Constant' *)
        i2_Chart_jj(ssMethodType := SS_OUTPUT, In := ContactorState_i, b_n := 5.0);
        rtb_IT_boUDC_EV_IsolationMeasurementRequest := i2_Chart_jj.Out;
        (* Outputs for Atomic SubSystem: '<Root>/ChiefMaster' *)
        (* Logic: '<S86>/AND' incorporates:
         *  Constant: '<S76>/Constant'
         *  Logic: '<S86>/AND2'
         *  RelationalOperator: '<S76>/Compare' *)
        i2_Chart1(ssMethodType := SS_OUTPUT, In := ((rtb_Switch2_k = 1.0) AND rtb_IT_boUDC_EV_IsolationMeasurementRequest) AND rtb_IT_boUDC_KL15_C);
        rtb_Out_ap := i2_Chart1.Out;
        (* Outputs for Atomic SubSystem: '<S676>/BatteryPackSignals' *)
        (* Logic: '<S12>/OR3' incorporates:
         *  Logic: '<S122>/AND'
         *  Logic: '<S12>/OR4'
         *  Logic: '<S12>/OR5'
         *  Logic: '<S12>/OR6'
         *  Logic: '<S12>/OR7'
         *  Logic: '<S12>/OR8'
         *  Logic: '<S12>/OR9'
         *  Outport: '<Root>/DO_KL15_BB1'
         *  Outport: '<Root>/DO_KL15_BB2'
         *  Outport: '<Root>/DO_KL15_BB3'
         *  SignalConversion: '<S682>/BusConversion_InsertedFor_IT_BatterySignal_Databus_at_inport_0'
         *  UnitDelay: '<S122>/Unit Delay7'
         *  UnitDelay: '<S122>/Unit Delay8'
         *  UnitDelay: '<S122>/Unit Delay9'
         *  UnitDelay: '<S12>/Unit Delay1'
         *  UnitDelay: '<S12>/Unit Delay4' *)
        i0_CMState(ssMethodType := SS_OUTPUT, KL15 := rtb_IT_boUDC_KL15_D OR rtb_IT_boUDC_KL15_C, KL15_AllBoxes := (DO_KL15_BB1 AND DO_KL15_BB2) AND DO_KL15_BB3, InsulationReadyOK := (rtb_S_in OR rtb_IP_boBatt1_Actia_Availability) OR rtb_Delay_dl, BattRelay_Closed := (rtb_IP_boBMS_HV_REL_ON_BB1 OR rtb_IP_boBMS_HV_REL_ON_BB2) OR rtb_IP_boBMS_HV_REL_ON_BB3, IMD_Available := (rtb_IP_boBMS_IMD_Active_BB1 OR rtb_IP_boBMS_IMD_Active_BB2) OR rtb_IP_boBMS_IMD_Active_BB3, BattRelay_Close_Req := ((REQ_HV_ON_a <> 0.0) OR (REQ_HV_ON_d <> 0.0)) OR (REQ_HV_ON <> 0.0), REQ_IMD_ON := (UnitDelay9_DSTATE_d AND UnitDelay8_DSTATE_k) AND UnitDelay7_DSTATE_h, FL_boREQ_MainHV_ON_MINUS := UnitDelay4_DSTATE_n, MainHV_Plus_Status := UnitDelay1_DSTATE_l, ShutdownError := rtb_Delay_j OR System_Error);
        CMState_e2 := i0_CMState.FL_u8SS_ChiefMaster_State;
        (* End of Outputs for SubSystem: '<S676>/BatteryPackSignals' *)
        (* End of Outputs for SubSystem: '<Root>/ChiefMaster' *)
        

        (* Outport: '<Root>/DO_boEMSRET_BB1_1' *)
        i0_EMSRET_Power(ssMethodType := SS_OUTPUT, ESD := rtb_Delay_j, HVILNOK := rtb_FL_boSS_HVIL_NOK, b_Reset := rtb_FL_boKL15_Reset);
        DO_boEMSRET_BB1_1 := i0_EMSRET_Power.FL_boSS_EMSRET_POWER;
        (* Outputs for Atomic SubSystem: '<Root>/ChiefMaster' *)
        (* Chart: '<S108>/Chart' incorporates:
         *  Constant: '<S108>/Constant2' *)
        (* Gateway: ChiefMaster/Flow Logic/System Status/AlarmBuzzer/Chart *)
        (* During: ChiefMaster/Flow Logic/System Status/AlarmBuzzer/Chart *)

        IF is_active_c49_ChiefMaster = 0 THEN 
            (* Entry: ChiefMaster/Flow Logic/System Status/AlarmBuzzer/Chart *)
            is_active_c49_ChiefMaster := 1;
            (* Entry Internal: ChiefMaster/Flow Logic/System Status/AlarmBuzzer/Chart *)
            (* Transition: '<S123>:2' *)
            is_c49_ChiefMaster := ChiefMaster_IN_BuzzerON;
            temporalCounter_i1(timerAction := 1, maxTime := 0);
            (* Entry 'BuzzerON': '<S123>:1' *)
            (* '<S123>:1:2' out=true; *)
            rtb_IT_boUDC_EV_IsolationMeasurementRequest := TRUE;
        ELSE 

            CASE is_c49_ChiefMaster OF
                ChiefMaster_IN_BuzzerOFF: 
                    (* During 'BuzzerOFF': '<S123>:3' *)
                    (* '<S123>:3:2' out=false; *)
                    rtb_IT_boUDC_EV_IsolationMeasurementRequest := FALSE;
                ELSE
                    (* During 'BuzzerON': '<S123>:1' *)
                    (* '<S123>:4:1' sf_internal_predicateOutput = after(BuzzerTimer,sec); *)
                    temporalCounter_i1(timerAction := 2, maxTime := USINT_TO_DINT(FL_u8HMI_BuzzerTimer) * 1000);

                    IF temporalCounter_i1.done THEN 
                        (* Transition: '<S123>:4' *)
                        is_c49_ChiefMaster := ChiefMaster_IN_BuzzerOFF;
                        (* Entry 'BuzzerOFF': '<S123>:3' *)
                        (* '<S123>:3:2' out=false; *)
                        rtb_IT_boUDC_EV_IsolationMeasurementRequest := FALSE;
                    ELSE 
                        (* '<S123>:1:2' out=true; *)
                        rtb_IT_boUDC_EV_IsolationMeasurementRequest := TRUE;
                    END_IF;

            END_CASE;

        END_IF;

        (* End of Chart: '<S108>/Chart' *)
        

        (* Switch: '<S108>/Switch' incorporates:
         *  Constant: '<S108>/Constant'
         *  Constant: '<S108>/Constant1'
         *  Logic: '<S108>/OR3' *)

        IF (System_Error OR rtb_Delay_j) OR rtb_IT_boUDC_EV_IsolationMeasurementRequest THEN 
            DO_CabinAlarm := TRUE;
        ELSE 
            DO_CabinAlarm := FALSE;
        END_IF;

        (* End of Switch: '<S108>/Switch' *)
        

        (* Outputs for Atomic SubSystem: '<S676>/BatteryPackSignals' *)
        (* Switch: '<S110>/Switch4' incorporates:
         *  SignalConversion: '<S682>/BusConversion_InsertedFor_IT_BatterySignal_Databus_at_inport_0' *)

        IF rtb_IP_boBMS_HV_REL_ON_BB1 THEN 
            rtb_Divide_h := rtb_Add_ic5;
        ELSE 
            rtb_Divide_h := rtb_FL_sSS_MaxDisChargeCurrent;
        END_IF;

        (* End of Switch: '<S110>/Switch4' *)
        

        (* Switch: '<S110>/Switch5' incorporates:
         *  SignalConversion: '<S682>/BusConversion_InsertedFor_IT_BatterySignal_Databus_at_inport_0' *)

        IF rtb_IP_boBMS_HV_REL_ON_BB2 THEN 
            rtb_Switch5_bs := rtb_Add_kf;
        ELSE 
            rtb_Switch5_bs := rtb_FL_sSS_MaxDisChargeCurrent;
        END_IF;

        (* End of Switch: '<S110>/Switch5' *)
        

        (* Switch: '<S110>/Switch6' incorporates:
         *  SignalConversion: '<S682>/BusConversion_InsertedFor_IT_BatterySignal_Databus_at_inport_0' *)

        IF rtb_IP_boBMS_HV_REL_ON_BB3 THEN 
            rtb_FL_sSS_MaxDisChargeCurrent := rtb_Add_j3;
        END_IF;

        (* End of Switch: '<S110>/Switch6' *)
        (* End of Outputs for SubSystem: '<S676>/BatteryPackSignals' *)
        

        (* Product: '<S110>/Product1' incorporates:
         *  MinMax: '<S110>/Min1'
         *  Sum: '<S110>/Add' *)

        IF rtb_NOT_m5 THEN 
            temp4 := MIN(rtb_Divide_h, rtb_Switch5_bs);
            temp3 := USINT_TO_REAL(rtb_ExtractDesiredBits_bk_tmp) * MIN(temp4, rtb_FL_sSS_MaxDisChargeCurrent);
        ELSE 
            temp3 := 0.0;
        END_IF;

        rtb_FL_sSS_MaxDisChargeCurrent := temp3;
        (* DiscretePulseGenerator: '<S114>/Discrete Pulse Generator20' *)
        Count_k := PLC_BOOL_TO_LREAL(in := (clockTickCounter < 50) AND (clockTickCounter >= 0));

        IF clockTickCounter >= 99 THEN 
            clockTickCounter := 0;
        ELSE 
            clockTickCounter := clockTickCounter + 1;
        END_IF;

        (* End of DiscretePulseGenerator: '<S114>/Discrete Pulse Generator20' *)
        

        (* Switch: '<S114>/Switch2' incorporates:
         *  Constant: '<S114>/Constant6'
         *  Switch: '<S114>/Switch'
         *  Switch: '<S114>/Switch1' *)

        IF rtb_boData_Out THEN 
            DO_boResetButton_LED := TRUE;
        ELSIF rtb_Delay_j THEN 
            (* Switch: '<S114>/Switch' incorporates:
             *  DataTypeConversion: '<S114>/Data Type Conversion30' *)
            DO_boResetButton_LED := Count_k <> 0.0;
        ELSE 
            (* Switch: '<S114>/Switch' incorporates:
             *  Constant: '<S114>/Constant1' *)
            DO_boResetButton_LED := FALSE;
        END_IF;

        (* End of Switch: '<S114>/Switch2' *)
        

        (* Outputs for Atomic SubSystem: '<S676>/BatteryPackSignals' *)
        (* Switch: '<S118>/Switch3' incorporates:
         *  Constant: '<S118>/Constant'
         *  Constant: '<S118>/Constant1'
         *  Logic: '<S118>/OR'
         *  SignalConversion: '<S682>/BusConversion_InsertedFor_IT_BatterySignal_Databus_at_inport_0' *)

        IF (rtb_IP_boBMS_HV_REL_ON_BB3 OR rtb_IP_boBMS_HV_REL_ON_BB2) OR rtb_IP_boBMS_HV_REL_ON_BB1 THEN 
            rtb_ExtractDesiredBits_be := NotAvailable_uint8;
        ELSE 
            rtb_ExtractDesiredBits_be := 0;
        END_IF;

        (* End of Switch: '<S118>/Switch3' *)
        

        (* Switch: '<S118>/Switch' incorporates:
         *  SignalConversion: '<S682>/BusConversion_InsertedFor_IT_BatterySignal_Databus_at_inport_0' *)

        IF rtb_IP_boBMS_HV_REL_ON_BB1 THEN 
            rtb_ExtractDesiredBits_mi := rtb_DataTypeConversion_k;
        ELSE 
            rtb_ExtractDesiredBits_mi := rtb_ExtractDesiredBits_be;
        END_IF;

        (* End of Switch: '<S118>/Switch' *)
        

        (* Switch: '<S118>/Switch1' incorporates:
         *  SignalConversion: '<S682>/BusConversion_InsertedFor_IT_BatterySignal_Databus_at_inport_0' *)

        IF rtb_IP_boBMS_HV_REL_ON_BB2 THEN 
            rtb_ExtractDesiredBits_ebk := rtb_DataTypeConversion1;
        ELSE 
            rtb_ExtractDesiredBits_ebk := rtb_ExtractDesiredBits_be;
        END_IF;

        (* End of Switch: '<S118>/Switch1' *)
        

        (* Switch: '<S118>/Switch2' incorporates:
         *  SignalConversion: '<S682>/BusConversion_InsertedFor_IT_BatterySignal_Databus_at_inport_0' *)

        IF rtb_IP_boBMS_HV_REL_ON_BB3 THEN 
            rtb_ExtractDesiredBits_be := rtb_DataTypeConversion2_h;
        END_IF;

        (* End of Switch: '<S118>/Switch2' *)
        (* End of Outputs for SubSystem: '<S676>/BatteryPackSignals' *)
        

        (* DataTypeConversion: '<S823>/Data Type Conversion1' *)
        v := ABS(Precharge_Satus);

        IF v < 4.503599627370496E+15 THEN 

            IF v >= 0.5 THEN 
                Count_k := rt_floord(u := Precharge_Satus + 0.5);
            ELSE 
                Count_k := 0.0;
            END_IF;

        ELSE 
            Count_k := Precharge_Satus;
        END_IF;

        (* DataTypeConversion: '<S823>/Data Type Conversion3' *)
        v := ABS(MainHV_Plus_Status);

        IF v < 4.503599627370496E+15 THEN 

            IF v >= 0.5 THEN 
                y := rt_floord(u := MainHV_Plus_Status + 0.5);
            ELSE 
                y := 0.0;
            END_IF;

        ELSE 
            y := MainHV_Plus_Status;
        END_IF;

        (* Outport: '<Root>/OP_ChiefMaster_BDU_Msg6' incorporates:
         *  ArithShift: '<S823>/Shift Arithmetic1'
         *  ArithShift: '<S823>/Shift Arithmetic3'
         *  DataTypeConversion: '<S820>/Extract Desired Bits'
         *  DataTypeConversion: '<S823>/Data Type Conversion1'
         *  DataTypeConversion: '<S823>/Data Type Conversion3'
         *  Sum: '<S823>/Add' *)
        OP_ChiefMaster_BDU_Msg6[5] := UDINT_TO_USINT(USINT_TO_UDINT(UDINT_TO_USINT(USINT_TO_UDINT(UDINT_TO_USINT(USINT_TO_UDINT(UDINT_TO_USINT(USINT_TO_UDINT(UDINT_TO_USINT(USINT_TO_UDINT(UDINT_TO_USINT(USINT_TO_UDINT(UDINT_TO_USINT(USINT_TO_UDINT(ShiftArithmetic6) + USINT_TO_UDINT(ShiftArithmetic5))) + USINT_TO_UDINT(ShiftArithmetic4))) + DINT_TO_UDINT(DWORD_TO_DINT(SHL(DINT_TO_DWORD(USINT_TO_DINT(WeldingDetection_Status)) AND 3, 4))))) + USINT_TO_UDINT(ShiftArithmetic2))) + USINT_TO_UDINT(BYTE_TO_USINT(SHL(USINT_TO_BYTE(DINT_TO_USINT(TRUNC(Count_k))), 2))))) + USINT_TO_UDINT(ShiftArithmetic))) + USINT_TO_UDINT(DINT_TO_USINT(TRUNC(y))));
        (* DataTypeConversion: '<S824>/Data Type Conversion1' *)

        IF rtb_UnitDelay2 >= 0.5 THEN 
            Count_k := rt_floord(u := rtb_UnitDelay2 + 0.5);
        ELSE 
            Count_k := 0.0;
        END_IF;

        (* DataTypeConversion: '<S824>/Data Type Conversion3' *)

        IF rtb_Uk1 >= 0.5 THEN 
            y := rt_floord(u := rtb_Uk1 + 0.5);
        ELSE 
            y := 0.0;
        END_IF;

        (* Outport: '<Root>/OP_ChiefMaster_BDU_Msg6' incorporates:
         *  ArithShift: '<S824>/Shift Arithmetic1'
         *  DataTypeConversion: '<S824>/Data Type Conversion1'
         *  DataTypeConversion: '<S824>/Data Type Conversion3'
         *  Sum: '<S824>/Add' *)
        OP_ChiefMaster_BDU_Msg6[6] := UDINT_TO_USINT(USINT_TO_UDINT(UDINT_TO_USINT(USINT_TO_UDINT(UDINT_TO_USINT(USINT_TO_UDINT(UDINT_TO_USINT(USINT_TO_UDINT(UDINT_TO_USINT(USINT_TO_UDINT(UDINT_TO_USINT(USINT_TO_UDINT(UDINT_TO_USINT(USINT_TO_UDINT(ShiftArithmetic6_a) + USINT_TO_UDINT(ShiftArithmetic5_j))) + USINT_TO_UDINT(ShiftArithmetic4_h))) + USINT_TO_UDINT(ShiftArithmetic3))) + USINT_TO_UDINT(ShiftArithmetic2_c))) + USINT_TO_UDINT(BYTE_TO_USINT(SHL(USINT_TO_BYTE(DINT_TO_USINT(TRUNC(Count_k))), 2))))) + USINT_TO_UDINT(ShiftArithmetic_n))) + DINT_TO_UDINT(TRUNC(y)));
        (* DataTypeConversion: '<S825>/Data Type Conversion6' *)
        v := ABS(MainHV_Minus_Status);

        IF v < 4.503599627370496E+15 THEN 

            IF v >= 0.5 THEN 
                Count_k := rt_floord(u := MainHV_Minus_Status + 0.5);
            ELSE 
                Count_k := 0.0;
            END_IF;

        ELSE 
            Count_k := MainHV_Minus_Status;
        END_IF;

        (* Outport: '<Root>/OP_ChiefMaster_BDU_Msg6' incorporates:
         *  ArithShift: '<S825>/Shift Arithmetic'
         *  ArithShift: '<S825>/Shift Arithmetic1'
         *  ArithShift: '<S825>/Shift Arithmetic2'
         *  ArithShift: '<S825>/Shift Arithmetic3'
         *  ArithShift: '<S825>/Shift Arithmetic4'
         *  ArithShift: '<S825>/Shift Arithmetic5'
         *  DataTypeConversion: '<S825>/Data Type Conversion'
         *  DataTypeConversion: '<S825>/Data Type Conversion1'
         *  DataTypeConversion: '<S825>/Data Type Conversion2'
         *  DataTypeConversion: '<S825>/Data Type Conversion3'
         *  DataTypeConversion: '<S825>/Data Type Conversion4'
         *  DataTypeConversion: '<S825>/Data Type Conversion5'
         *  DataTypeConversion: '<S825>/Data Type Conversion6'
         *  Sum: '<S825>/Add' *)
        OP_ChiefMaster_BDU_Msg6[4] := UDINT_TO_USINT(USINT_TO_UDINT(UDINT_TO_USINT(USINT_TO_UDINT(UDINT_TO_USINT(USINT_TO_UDINT(UDINT_TO_USINT(USINT_TO_UDINT(UDINT_TO_USINT(USINT_TO_UDINT(UDINT_TO_USINT(USINT_TO_UDINT(UDINT_TO_USINT(USINT_TO_UDINT(BYTE_TO_USINT(SHL(USINT_TO_BYTE(DINT_TO_USINT(TRUNC(Count_k))), 6))) + USINT_TO_UDINT(ShiftArithmetic6_f))) + DINT_TO_UDINT(DWORD_TO_DINT(SHL(DINT_TO_DWORD(BOOL_TO_DINT(rtb_Out_k)), 5))))) + DINT_TO_UDINT(DWORD_TO_DINT(SHL(DINT_TO_DWORD(BOOL_TO_DINT(MainHV_Plus_Welded)), 4))))) + DINT_TO_UDINT(DWORD_TO_DINT(SHL(DINT_TO_DWORD(BOOL_TO_DINT(MainHV_Minus_Welded)), 3))))) + DINT_TO_UDINT(DWORD_TO_DINT(SHL(DINT_TO_DWORD(BOOL_TO_DINT(DO_REQ_MainHV_ON_PLUS)), 2))))) + DINT_TO_UDINT(DWORD_TO_DINT(SHL(DINT_TO_DWORD(BOOL_TO_DINT(DO_REQ_MainHV_ON_Precharge)), 1))))) + BOOL_TO_UDINT(DO_REQ_MainHV_ON_MINUS));
        (* Product: '<S833>/Divide' incorporates:
         *  Constant: '<S826>/Constant1'
         *  Sum: '<S833>/Add' *)
        rtb_UnitDelay := rtb_Divide_i / 0.1;
        (* DataTypeConversion: '<S832>/Data Type Conversion2' *)
        rtb_Divide_h := ABS(rtb_UnitDelay);

        IF rtb_Divide_h < 8.388608E+6 THEN 

            IF rtb_Divide_h >= 0.5 THEN 
                rtb_UnitDelay := rt_floorf(u := rtb_UnitDelay + 0.5);
            ELSE 
                rtb_UnitDelay := 0.0;
            END_IF;

        END_IF;

        (* Product: '<S837>/Divide' incorporates:
         *  Constant: '<S827>/Constant1'
         *  Sum: '<S837>/Add' *)
        rtb_Abs := rtb_Abs / 0.1;
        (* DataTypeConversion: '<S836>/Data Type Conversion2' *)
        rtb_Divide_h := ABS(rtb_Abs);

        IF rtb_Divide_h < 8.388608E+6 THEN 

            IF rtb_Divide_h >= 0.5 THEN 
                rtb_Abs := rt_floorf(u := rtb_Abs + 0.5);
            ELSE 
                rtb_Abs := 0.0;
            END_IF;

        END_IF;

        (* Product: '<S841>/Divide' incorporates:
         *  Constant: '<S828>/Constant1'
         *  Sum: '<S841>/Add' *)
        rtb_Abs1 := rtb_Abs1 / 0.1;
        (* DataTypeConversion: '<S840>/Data Type Conversion2' *)
        rtb_Divide_h := ABS(rtb_Abs1);

        IF rtb_Divide_h < 8.388608E+6 THEN 

            IF rtb_Divide_h >= 0.5 THEN 
                rtb_Abs1 := rt_floorf(u := rtb_Abs1 + 0.5);
            ELSE 
                rtb_Abs1 := 0.0;
            END_IF;

        END_IF;

        (* Product: '<S845>/Divide' incorporates:
         *  Constant: '<S829>/Constant1'
         *  Sum: '<S845>/Add' *)
        rtb_Abs2 := rtb_Abs2 / 0.1;
        (* DataTypeConversion: '<S844>/Data Type Conversion2' *)
        rtb_Divide_h := ABS(rtb_Abs2);

        IF rtb_Divide_h < 8.388608E+6 THEN 

            IF rtb_Divide_h >= 0.5 THEN 
                rtb_Abs2 := rt_floorf(u := rtb_Abs2 + 0.5);
            ELSE 
                rtb_Abs2 := 0.0;
            END_IF;

        END_IF;

        (* Product: '<S849>/Divide' incorporates:
         *  Constant: '<S830>/Constant1'
         *  Sum: '<S849>/Add' *)
        rtb_Divide1_p := rtb_Divide1_p / 0.1;
        (* DataTypeConversion: '<S848>/Data Type Conversion2' *)
        rtb_Divide_h := ABS(rtb_Divide1_p);

        IF rtb_Divide_h < 8.388608E+6 THEN 

            IF rtb_Divide_h >= 0.5 THEN 
                rtb_Divide1_p := rt_floorf(u := rtb_Divide1_p + 0.5);
            ELSE 
                rtb_Divide1_p := 0.0;
            END_IF;

        END_IF;

        (* Product: '<S853>/Divide' incorporates:
         *  Constant: '<S831>/Constant1'
         *  Sum: '<S853>/Add' *)
        rtb_Divide2 := rtb_Divide2 / 0.1;
        (* DataTypeConversion: '<S852>/Data Type Conversion2' *)
        rtb_Divide_h := ABS(rtb_Divide2);

        IF rtb_Divide_h < 8.388608E+6 THEN 

            IF rtb_Divide_h >= 0.5 THEN 
                rtb_Divide2 := rt_floorf(u := rtb_Divide2 + 0.5);
            ELSE 
                rtb_Divide2 := 0.0;
            END_IF;

        END_IF;

        (* Outputs for Atomic SubSystem: '<S676>/BatteryPackSignals' *)
        (* Product: '<S862>/Divide' incorporates:
         *  Constant: '<S804>/Constant2'
         *  SignalConversion: '<S682>/BusConversion_InsertedFor_IT_BatterySignal_Databus_at_inport_0' *)
        rtb_Min := rtb_Min / 0.1;
        (* End of Outputs for SubSystem: '<S676>/BatteryPackSignals' *)
        

        (* DataTypeConversion: '<S858>/Data Type Conversion2' *)

        IF rtb_Min >= 0.5 THEN 
            rtb_Switch3 := rt_floorf(u := rtb_Min + 0.5);
        ELSE 
            rtb_Switch3 := 0.0;
        END_IF;

        (* Outputs for Atomic SubSystem: '<S676>/BatteryPackSignals' *)
        (* Product: '<S863>/Divide' incorporates:
         *  Constant: '<S804>/Constant3'
         *  SignalConversion: '<S682>/BusConversion_InsertedFor_IT_BatterySignal_Databus_at_inport_0' *)
        rtb_Min := rtb_Add_ki5 / 0.1;
        (* End of Outputs for SubSystem: '<S676>/BatteryPackSignals' *)
        

        (* DataTypeConversion: '<S859>/Data Type Conversion2' *)

        IF ABS(rtb_Min) >= 0.5 THEN 
            rtb_Switch_a := rt_floorf(u := rtb_Min + 0.5);
        ELSE 
            rtb_Switch_a := 0.0;
        END_IF;

        (* MultiPortSwitch: '<S1049>/Multiport Switch' incorporates:
         *  Constant: '<S1049>/Constant' *)

        CASE TRUNC(rtb_BattSelect_f) OF
            1: 
                DO_boKL15_IMD_BB1 := rtb_IT_boChargeStop_Button;
            2: 
                DO_boKL15_IMD_BB1 := rtb_IT_boChargeStop_Button;
            3: 
                DO_boKL15_IMD_BB1 := FALSE;
            ELSE
                DO_boKL15_IMD_BB1 := FALSE;
        END_CASE;

        (* End of MultiPortSwitch: '<S1049>/Multiport Switch' *)
        

        (* DataTypeConversion: '<S860>/Data Type Conversion5' *)
        v := ABS(rtb_Contactor_FB_State_h);

        IF v < 4.503599627370496E+15 THEN 

            IF v >= 0.5 THEN 
                Count_k := rt_floord(u := rtb_Contactor_FB_State_h + 0.5);
            ELSE 
                Count_k := 0.0;
            END_IF;

        ELSE 
            Count_k := rtb_Contactor_FB_State_h;
        END_IF;

        (* DataTypeConversion: '<S860>/Data Type Conversion4' incorporates:
         *  DataTypeConversion: '<S1020>/Data Type Conversion3'
         *  DataTypeConversion: '<S1031>/Data Type Conversion1'
         *  DataTypeConversion: '<S981>/Data Type Conversion' *)
        rtb_Uk1 := ABS(REQ_HV_ON_a);

        IF rtb_Uk1 < 4.503599627370496E+15 THEN 

            IF rtb_Uk1 >= 0.5 THEN 
                y := rt_floord(u := REQ_HV_ON_a + 0.5);
            ELSE 
                y := 0.0;
            END_IF;

        ELSE 
            y := REQ_HV_ON_a;
        END_IF;

        (* DataTypeConversion: '<S860>/Data Type Conversion1' *)
        v := ABS(ContactorState_i);

        IF v < 4.503599627370496E+15 THEN 

            IF v >= 0.5 THEN 
                v := rt_floord(u := ContactorState_i + 0.5);
            ELSE 
                v := 0.0;
            END_IF;

        ELSE 
            v := ContactorState_i;
        END_IF;

        (* Outputs for Atomic SubSystem: '<S676>/BatteryPackSignals' *)
        (* DataTypeConversion: '<S860>/Data Type Conversion3' incorporates:
         *  SignalConversion: '<S682>/BusConversion_InsertedFor_IT_BatterySignal_Databus_at_inport_0' *)

        IF DINT_TO_LREAL(rtb_IP_boBMS_Batt1_Availability) >= 0.5 THEN 
            y_0 := rt_floord(u := DINT_TO_LREAL(rtb_IP_boBMS_Batt1_Availability) + 0.5);
        ELSE 
            y_0 := 0.0;
        END_IF;

        (* End of Outputs for SubSystem: '<S676>/BatteryPackSignals' *)
        

        (* Sum: '<S860>/Add' incorporates:
         *  ArithShift: '<S860>/Shift Arithmetic'
         *  DataTypeConversion: '<S860>/Data Type Conversion'
         *  Sum: '<S1020>/Add' *)
        OP_ChiefMaster_Battery1_Msg7_tmp := DINT_TO_UDINT(DWORD_TO_DINT(SHL(DINT_TO_DWORD(BOOL_TO_DINT(DO_boKL15_IMD_BB1)), 1)));
        (* Outputs for Atomic SubSystem: '<S676>/BatteryPackSignals' *)
        (* Outport: '<Root>/OP_ChiefMaster_Battery1_Msg7' incorporates:
         *  ArithShift: '<S860>/Shift Arithmetic1'
         *  ArithShift: '<S860>/Shift Arithmetic3'
         *  ArithShift: '<S860>/Shift Arithmetic4'
         *  ArithShift: '<S860>/Shift Arithmetic6'
         *  DataTypeConversion: '<S860>/Data Type Conversion1'
         *  DataTypeConversion: '<S860>/Data Type Conversion3'
         *  DataTypeConversion: '<S860>/Data Type Conversion4'
         *  DataTypeConversion: '<S860>/Data Type Conversion5'
         *  DataTypeConversion: '<S860>/Data Type Conversion7'
         *  SignalConversion: '<S698>/Signal Copy'
         *  Sum: '<S860>/Add' *)
        OP_ChiefMaster_Battery1_Msg7[0] := UDINT_TO_USINT(USINT_TO_UDINT(UDINT_TO_USINT(USINT_TO_UDINT(UDINT_TO_USINT(USINT_TO_UDINT(UDINT_TO_USINT(USINT_TO_UDINT(UDINT_TO_USINT(USINT_TO_UDINT(UDINT_TO_USINT(USINT_TO_UDINT(UDINT_TO_USINT(DINT_TO_UDINT(DWORD_TO_DINT(SHL(DINT_TO_DWORD(BOOL_TO_DINT(rtb_IP_boBMS_SDError_BB1)), 7))) + USINT_TO_UDINT(ShiftArithmetic5_h))) + USINT_TO_UDINT(BYTE_TO_USINT(SHL(USINT_TO_BYTE(DINT_TO_USINT(TRUNC(Count_k))), 5))))) + USINT_TO_UDINT(BYTE_TO_USINT(SHL(USINT_TO_BYTE(DINT_TO_USINT(TRUNC(y))), 4))))) + USINT_TO_UDINT(ShiftArithmetic2_o))) + USINT_TO_UDINT(BYTE_TO_USINT(SHL(USINT_TO_BYTE(DINT_TO_USINT(TRUNC(v))), 2))))) + OP_ChiefMaster_Battery1_Msg7_tmp)) + DINT_TO_UDINT(TRUNC(y_0)));
        (* Product: '<S872>/Divide' incorporates:
         *  Constant: '<S805>/Constant4'
         *  SignalConversion: '<S682>/BusConversion_InsertedFor_IT_BatterySignal_Databus_at_inport_0' *)
        rtb_Min := rtb_Add_ic5 / 0.1;
        (* End of Outputs for SubSystem: '<S676>/BatteryPackSignals' *)
        

        (* DataTypeConversion: '<S868>/Data Type Conversion2' *)

        IF rtb_Min >= 0.5 THEN 
            rtb_Add_ic5 := rt_floorf(u := rtb_Min + 0.5);
        ELSE 
            rtb_Add_ic5 := 0.0;
        END_IF;

        (* Outputs for Atomic SubSystem: '<S676>/BatteryPackSignals' *)
        (* Product: '<S873>/Divide' incorporates:
         *  Constant: '<S805>/Constant3'
         *  SignalConversion: '<S682>/BusConversion_InsertedFor_IT_BatterySignal_Databus_at_inport_0' *)
        rtb_Min := rtb_Add_b / 0.1;
        (* End of Outputs for SubSystem: '<S676>/BatteryPackSignals' *)
        

        (* DataTypeConversion: '<S869>/Data Type Conversion2' *)

        IF rtb_Min >= 0.5 THEN 
            rtb_Add_b := rt_floorf(u := rtb_Min + 0.5);
        ELSE 
            rtb_Add_b := 0.0;
        END_IF;

        (* Outputs for Atomic SubSystem: '<S676>/BatteryPackSignals' *)
        (* Product: '<S874>/Divide' incorporates:
         *  Constant: '<S805>/Constant6'
         *  SignalConversion: '<S682>/BusConversion_InsertedFor_IT_BatterySignal_Databus_at_inport_0' *)
        rtb_Min := rtb_Add_cv / 100.0;
        (* End of Outputs for SubSystem: '<S676>/BatteryPackSignals' *)
        

        (* DataTypeConversion: '<S870>/Data Type Conversion2' *)
        rtb_Divide_h := ABS(rtb_Min);

        IF rtb_Divide_h < 8.388608E+6 THEN 

            IF rtb_Divide_h >= 0.5 THEN 
                rtb_Min := rt_floorf(u := rtb_Min + 0.5);
            ELSE 
                rtb_Min := 0.0;
            END_IF;

        END_IF;

        (* Outputs for Atomic SubSystem: '<S676>/BatteryPackSignals' *)
        (* Product: '<S875>/Divide' incorporates:
         *  Constant: '<S805>/Constant8'
         *  SignalConversion: '<S682>/BusConversion_InsertedFor_IT_BatterySignal_Databus_at_inport_0' *)
        rtb_Add_psl := rtb_Add_psl / 100.0;
        (* End of Outputs for SubSystem: '<S676>/BatteryPackSignals' *)
        

        (* DataTypeConversion: '<S871>/Data Type Conversion2' *)
        rtb_Divide_h := ABS(rtb_Add_psl);

        IF rtb_Divide_h < 8.388608E+6 THEN 

            IF rtb_Divide_h >= 0.5 THEN 
                rtb_Add_psl := rt_floorf(u := rtb_Add_psl + 0.5);
            ELSE 
                rtb_Add_psl := 0.0;
            END_IF;

        END_IF;

        (* Outputs for Atomic SubSystem: '<S676>/BatteryPackSignals' *)
        (* Product: '<S888>/Divide' incorporates:
         *  Constant: '<S806>/Constant6'
         *  SignalConversion: '<S682>/BusConversion_InsertedFor_IT_BatterySignal_Databus_at_inport_0' *)
        rtb_Add_cv := rtb_Add_nm / 0.1;
        (* End of Outputs for SubSystem: '<S676>/BatteryPackSignals' *)
        

        (* DataTypeConversion: '<S884>/Data Type Conversion2' *)

        IF rtb_Add_cv >= 0.5 THEN 
            rtb_Switch2_k := rt_floorf(u := rtb_Add_cv + 0.5);
        ELSE 
            rtb_Switch2_k := 0.0;
        END_IF;

        (* Outputs for Atomic SubSystem: '<S676>/BatteryPackSignals' *)
        (* Product: '<S889>/Divide' incorporates:
         *  Constant: '<S806>/Constant8'
         *  SignalConversion: '<S682>/BusConversion_InsertedFor_IT_BatterySignal_Databus_at_inport_0' *)
        rtb_Add_cv := rtb_Add_ie / 0.1;
        (* End of Outputs for SubSystem: '<S676>/BatteryPackSignals' *)
        

        (* DataTypeConversion: '<S885>/Data Type Conversion2' *)

        IF rtb_Add_cv >= 0.5 THEN 
            rtb_Add_ie := rt_floorf(u := rtb_Add_cv + 0.5);
        ELSE 
            rtb_Add_ie := 0.0;
        END_IF;

        (* Outputs for Atomic SubSystem: '<S676>/BatteryPackSignals' *)
        (* Product: '<S900>/Divide' incorporates:
         *  Constant: '<S807>/Constant2'
         *  SignalConversion: '<S682>/BusConversion_InsertedFor_IT_BatterySignal_Databus_at_inport_0' *)
        rtb_Add_cv := rtb_Add_an / 0.1;
        (* End of Outputs for SubSystem: '<S676>/BatteryPackSignals' *)
        

        (* DataTypeConversion: '<S896>/Data Type Conversion2' *)

        IF rtb_Add_cv >= 0.5 THEN 
            rtb_Add_an := rt_floorf(u := rtb_Add_cv + 0.5);
        ELSE 
            rtb_Add_an := 0.0;
        END_IF;

        (* Outputs for Atomic SubSystem: '<S676>/BatteryPackSignals' *)
        (* Product: '<S901>/Divide' incorporates:
         *  Constant: '<S807>/Constant3'
         *  SignalConversion: '<S682>/BusConversion_InsertedFor_IT_BatterySignal_Databus_at_inport_0' *)
        rtb_Add_cv := rtb_Add_ir / 0.1;
        (* End of Outputs for SubSystem: '<S676>/BatteryPackSignals' *)
        

        (* DataTypeConversion: '<S897>/Data Type Conversion2' *)

        IF ABS(rtb_Add_cv) >= 0.5 THEN 
            rtb_Add_ci := rt_floorf(u := rtb_Add_cv + 0.5);
        ELSE 
            rtb_Add_ci := 0.0;
        END_IF;

        (* MultiPortSwitch: '<S1050>/Multiport Switch' incorporates:
         *  Constant: '<S1050>/Constant' *)

        CASE TRUNC(rtb_BattSelect) OF
            1: 
                DO_boKL15_IMD_BB2 := rtb_UnitDelay1_d;
            2: 
                DO_boKL15_IMD_BB2 := rtb_UnitDelay1_d;
            3: 
                DO_boKL15_IMD_BB2 := FALSE;
            ELSE
                DO_boKL15_IMD_BB2 := FALSE;
        END_CASE;

        (* End of MultiPortSwitch: '<S1050>/Multiport Switch' *)
        

        (* DataTypeConversion: '<S898>/Data Type Conversion5' *)
        v := ABS(rtb_Contactor_FB_State_g);

        IF v < 4.503599627370496E+15 THEN 

            IF v >= 0.5 THEN 
                Count_k := rt_floord(u := rtb_Contactor_FB_State_g + 0.5);
            ELSE 
                Count_k := 0.0;
            END_IF;

        ELSE 
            Count_k := rtb_Contactor_FB_State_g;
        END_IF;

        (* DataTypeConversion: '<S898>/Data Type Conversion4' incorporates:
         *  DataTypeConversion: '<S1021>/Data Type Conversion3'
         *  DataTypeConversion: '<S1037>/Data Type Conversion1'
         *  DataTypeConversion: '<S981>/Data Type Conversion1' *)
        rtb_UnitDelay2 := ABS(REQ_HV_ON_d);

        IF rtb_UnitDelay2 < 4.503599627370496E+15 THEN 

            IF rtb_UnitDelay2 >= 0.5 THEN 
                y := rt_floord(u := REQ_HV_ON_d + 0.5);
            ELSE 
                y := 0.0;
            END_IF;

        ELSE 
            y := REQ_HV_ON_d;
        END_IF;

        (* DataTypeConversion: '<S898>/Data Type Conversion1' *)
        v := ABS(ContactorState_f);

        IF v < 4.503599627370496E+15 THEN 

            IF v >= 0.5 THEN 
                v := rt_floord(u := ContactorState_f + 0.5);
            ELSE 
                v := 0.0;
            END_IF;

        ELSE 
            v := ContactorState_f;
        END_IF;

        (* Outputs for Atomic SubSystem: '<S676>/BatteryPackSignals' *)
        (* DataTypeConversion: '<S898>/Data Type Conversion3' incorporates:
         *  SignalConversion: '<S682>/BusConversion_InsertedFor_IT_BatterySignal_Databus_at_inport_0' *)

        IF DINT_TO_LREAL(rtb_UnitDelay5) >= 0.5 THEN 
            y_0 := rt_floord(u := DINT_TO_LREAL(rtb_UnitDelay5) + 0.5);
        ELSE 
            y_0 := 0.0;
        END_IF;

        (* End of Outputs for SubSystem: '<S676>/BatteryPackSignals' *)
        

        (* Sum: '<S898>/Add' incorporates:
         *  ArithShift: '<S898>/Shift Arithmetic'
         *  DataTypeConversion: '<S898>/Data Type Conversion'
         *  Sum: '<S1021>/Add' *)
        OP_ChiefMaster_Battery2_Msg10_tmp := DINT_TO_UDINT(DWORD_TO_DINT(SHL(DINT_TO_DWORD(BOOL_TO_DINT(DO_boKL15_IMD_BB2)), 1)));
        (* Outputs for Atomic SubSystem: '<S676>/BatteryPackSignals' *)
        (* Outport: '<Root>/OP_ChiefMaster_Battery2_Msg10' incorporates:
         *  ArithShift: '<S898>/Shift Arithmetic1'
         *  ArithShift: '<S898>/Shift Arithmetic3'
         *  ArithShift: '<S898>/Shift Arithmetic4'
         *  ArithShift: '<S898>/Shift Arithmetic6'
         *  DataTypeConversion: '<S898>/Data Type Conversion1'
         *  DataTypeConversion: '<S898>/Data Type Conversion3'
         *  DataTypeConversion: '<S898>/Data Type Conversion4'
         *  DataTypeConversion: '<S898>/Data Type Conversion5'
         *  DataTypeConversion: '<S898>/Data Type Conversion7'
         *  SignalConversion: '<S699>/Signal Copy'
         *  Sum: '<S898>/Add' *)
        OP_ChiefMaster_Battery2_Msg10[0] := UDINT_TO_USINT(USINT_TO_UDINT(UDINT_TO_USINT(USINT_TO_UDINT(UDINT_TO_USINT(USINT_TO_UDINT(UDINT_TO_USINT(USINT_TO_UDINT(UDINT_TO_USINT(USINT_TO_UDINT(UDINT_TO_USINT(USINT_TO_UDINT(UDINT_TO_USINT(DINT_TO_UDINT(DWORD_TO_DINT(SHL(DINT_TO_DWORD(BOOL_TO_DINT(rtb_IP_boBMS_SDError_BB2)), 7))) + USINT_TO_UDINT(ShiftArithmetic5_jh))) + USINT_TO_UDINT(BYTE_TO_USINT(SHL(USINT_TO_BYTE(DINT_TO_USINT(TRUNC(Count_k))), 5))))) + USINT_TO_UDINT(BYTE_TO_USINT(SHL(USINT_TO_BYTE(DINT_TO_USINT(TRUNC(y))), 4))))) + USINT_TO_UDINT(ShiftArithmetic2_n))) + USINT_TO_UDINT(BYTE_TO_USINT(SHL(USINT_TO_BYTE(DINT_TO_USINT(TRUNC(v))), 2))))) + OP_ChiefMaster_Battery2_Msg10_tmp)) + DINT_TO_UDINT(TRUNC(y_0)));
        (* Product: '<S910>/Divide' incorporates:
         *  Constant: '<S808>/Constant4'
         *  SignalConversion: '<S682>/BusConversion_InsertedFor_IT_BatterySignal_Databus_at_inport_0' *)
        rtb_Add_cv := rtb_Add_kf / 0.1;
        (* End of Outputs for SubSystem: '<S676>/BatteryPackSignals' *)
        

        (* DataTypeConversion: '<S906>/Data Type Conversion2' *)

        IF rtb_Add_cv >= 0.5 THEN 
            rtb_Add_kf := rt_floorf(u := rtb_Add_cv + 0.5);
        ELSE 
            rtb_Add_kf := 0.0;
        END_IF;

        (* Outputs for Atomic SubSystem: '<S676>/BatteryPackSignals' *)
        (* Product: '<S911>/Divide' incorporates:
         *  Constant: '<S808>/Constant3'
         *  SignalConversion: '<S682>/BusConversion_InsertedFor_IT_BatterySignal_Databus_at_inport_0' *)
        rtb_Add_cv := rtb_Add_h / 0.1;
        (* End of Outputs for SubSystem: '<S676>/BatteryPackSignals' *)
        

        (* DataTypeConversion: '<S907>/Data Type Conversion2' *)

        IF rtb_Add_cv >= 0.5 THEN 
            rtb_Add_h := rt_floorf(u := rtb_Add_cv + 0.5);
        ELSE 
            rtb_Add_h := 0.0;
        END_IF;

        (* Outputs for Atomic SubSystem: '<S676>/BatteryPackSignals' *)
        (* Product: '<S912>/Divide' incorporates:
         *  Constant: '<S808>/Constant6'
         *  SignalConversion: '<S682>/BusConversion_InsertedFor_IT_BatterySignal_Databus_at_inport_0' *)
        rtb_Add_cv := rtb_Add_d / 100.0;
        (* End of Outputs for SubSystem: '<S676>/BatteryPackSignals' *)
        

        (* DataTypeConversion: '<S908>/Data Type Conversion2' *)
        rtb_Divide_h := ABS(rtb_Add_cv);

        IF rtb_Divide_h < 8.388608E+6 THEN 

            IF rtb_Divide_h >= 0.5 THEN 
                rtb_Add_cv := rt_floorf(u := rtb_Add_cv + 0.5);
            ELSE 
                rtb_Add_cv := 0.0;
            END_IF;

        END_IF;

        (* Outputs for Atomic SubSystem: '<S676>/BatteryPackSignals' *)
        (* Product: '<S913>/Divide' incorporates:
         *  Constant: '<S808>/Constant8'
         *  SignalConversion: '<S682>/BusConversion_InsertedFor_IT_BatterySignal_Databus_at_inport_0' *)
        rtb_Add_ic := rtb_Add_ic / 100.0;
        (* End of Outputs for SubSystem: '<S676>/BatteryPackSignals' *)
        

        (* DataTypeConversion: '<S909>/Data Type Conversion2' *)
        rtb_Divide_h := ABS(rtb_Add_ic);

        IF rtb_Divide_h < 8.388608E+6 THEN 

            IF rtb_Divide_h >= 0.5 THEN 
                rtb_Add_ic := rt_floorf(u := rtb_Add_ic + 0.5);
            ELSE 
                rtb_Add_ic := 0.0;
            END_IF;

        END_IF;

        (* Outputs for Atomic SubSystem: '<S676>/BatteryPackSignals' *)
        (* Product: '<S926>/Divide' incorporates:
         *  Constant: '<S809>/Constant6'
         *  SignalConversion: '<S682>/BusConversion_InsertedFor_IT_BatterySignal_Databus_at_inport_0' *)
        rtb_Add_d := rtb_Add_d4 / 0.1;
        (* End of Outputs for SubSystem: '<S676>/BatteryPackSignals' *)
        

        (* DataTypeConversion: '<S922>/Data Type Conversion2' *)

        IF rtb_Add_d >= 0.5 THEN 
            rtb_Divide_i := rt_floorf(u := rtb_Add_d + 0.5);
        ELSE 
            rtb_Divide_i := 0.0;
        END_IF;

        (* Outputs for Atomic SubSystem: '<S676>/BatteryPackSignals' *)
        (* Product: '<S927>/Divide' incorporates:
         *  Constant: '<S809>/Constant8'
         *  SignalConversion: '<S682>/BusConversion_InsertedFor_IT_BatterySignal_Databus_at_inport_0' *)
        rtb_Add_d := rtb_Add_oy / 0.1;
        (* End of Outputs for SubSystem: '<S676>/BatteryPackSignals' *)
        

        (* DataTypeConversion: '<S923>/Data Type Conversion2' *)

        IF rtb_Add_d >= 0.5 THEN 
            rtb_Add_oy := rt_floorf(u := rtb_Add_d + 0.5);
        ELSE 
            rtb_Add_oy := 0.0;
        END_IF;

        (* Outputs for Atomic SubSystem: '<S676>/BatteryPackSignals' *)
        (* Product: '<S938>/Divide' incorporates:
         *  Constant: '<S810>/Constant2'
         *  SignalConversion: '<S682>/BusConversion_InsertedFor_IT_BatterySignal_Databus_at_inport_0' *)
        rtb_Add_d := rtb_Add_e / 0.1;
        (* End of Outputs for SubSystem: '<S676>/BatteryPackSignals' *)
        

        (* DataTypeConversion: '<S934>/Data Type Conversion2' *)

        IF rtb_Add_d >= 0.5 THEN 
            rtb_Add_e := rt_floorf(u := rtb_Add_d + 0.5);
        ELSE 
            rtb_Add_e := 0.0;
        END_IF;

        (* Outputs for Atomic SubSystem: '<S676>/BatteryPackSignals' *)
        (* Product: '<S939>/Divide' incorporates:
         *  Constant: '<S810>/Constant3'
         *  SignalConversion: '<S682>/BusConversion_InsertedFor_IT_BatterySignal_Databus_at_inport_0' *)
        rtb_Add_d := rtb_Add_m / 0.1;
        (* End of Outputs for SubSystem: '<S676>/BatteryPackSignals' *)
        

        (* DataTypeConversion: '<S935>/Data Type Conversion2' *)

        IF ABS(rtb_Add_d) >= 0.5 THEN 
            rtb_Switch5_bs := rt_floorf(u := rtb_Add_d + 0.5);
        ELSE 
            rtb_Switch5_bs := 0.0;
        END_IF;

        (* MultiPortSwitch: '<S1051>/Multiport Switch' incorporates:
         *  Constant: '<S1051>/Constant' *)

        CASE TRUNC(rtb_BattSelect_i) OF
            1: 
                DO_boKL15_IMD_BB3 := rtb_Out_bl;
            2: 
                DO_boKL15_IMD_BB3 := rtb_Out_bl;
            3: 
                DO_boKL15_IMD_BB3 := FALSE;
            ELSE
                DO_boKL15_IMD_BB3 := FALSE;
        END_CASE;

        (* End of MultiPortSwitch: '<S1051>/Multiport Switch' *)
        

        (* DataTypeConversion: '<S937>/Data Type Conversion5' *)
        v := ABS(rtb_Contactor_FB_State);

        IF v < 4.503599627370496E+15 THEN 

            IF v >= 0.5 THEN 
                Count_k := rt_floord(u := rtb_Contactor_FB_State + 0.5);
            ELSE 
                Count_k := 0.0;
            END_IF;

        ELSE 
            Count_k := rtb_Contactor_FB_State;
        END_IF;

        (* DataTypeConversion: '<S937>/Data Type Conversion4' incorporates:
         *  DataTypeConversion: '<S1022>/Data Type Conversion3'
         *  DataTypeConversion: '<S1043>/Data Type Conversion1'
         *  DataTypeConversion: '<S981>/Data Type Conversion2' *)
        v_tmp := ABS(REQ_HV_ON);

        IF v_tmp < 4.503599627370496E+15 THEN 

            IF v_tmp >= 0.5 THEN 
                y := rt_floord(u := REQ_HV_ON + 0.5);
            ELSE 
                y := 0.0;
            END_IF;

        ELSE 
            y := REQ_HV_ON;
        END_IF;

        (* DataTypeConversion: '<S937>/Data Type Conversion1' *)
        v := ABS(ContactorState);

        IF v < 4.503599627370496E+15 THEN 

            IF v >= 0.5 THEN 
                v := rt_floord(u := ContactorState + 0.5);
            ELSE 
                v := 0.0;
            END_IF;

        ELSE 
            v := ContactorState;
        END_IF;

        (* Outputs for Atomic SubSystem: '<S676>/BatteryPackSignals' *)
        (* DataTypeConversion: '<S937>/Data Type Conversion3' incorporates:
         *  SignalConversion: '<S682>/BusConversion_InsertedFor_IT_BatterySignal_Databus_at_inport_0' *)

        IF DINT_TO_LREAL(rtb_IP_boBMS_Batt3_Availability) >= 0.5 THEN 
            y_0 := rt_floord(u := DINT_TO_LREAL(rtb_IP_boBMS_Batt3_Availability) + 0.5);
        ELSE 
            y_0 := 0.0;
        END_IF;

        (* End of Outputs for SubSystem: '<S676>/BatteryPackSignals' *)
        

        (* Sum: '<S937>/Add' incorporates:
         *  ArithShift: '<S937>/Shift Arithmetic'
         *  DataTypeConversion: '<S937>/Data Type Conversion'
         *  Sum: '<S1022>/Add' *)
        OP_ChiefMaster_Battery3_Msg13_tmp := DINT_TO_UDINT(DWORD_TO_DINT(SHL(DINT_TO_DWORD(BOOL_TO_DINT(DO_boKL15_IMD_BB3)), 1)));
        (* Outputs for Atomic SubSystem: '<S676>/BatteryPackSignals' *)
        (* Outport: '<Root>/OP_ChiefMaster_Battery3_Msg13' incorporates:
         *  ArithShift: '<S937>/Shift Arithmetic1'
         *  ArithShift: '<S937>/Shift Arithmetic3'
         *  ArithShift: '<S937>/Shift Arithmetic4'
         *  ArithShift: '<S937>/Shift Arithmetic6'
         *  DataTypeConversion: '<S937>/Data Type Conversion1'
         *  DataTypeConversion: '<S937>/Data Type Conversion3'
         *  DataTypeConversion: '<S937>/Data Type Conversion4'
         *  DataTypeConversion: '<S937>/Data Type Conversion5'
         *  DataTypeConversion: '<S937>/Data Type Conversion7'
         *  SignalConversion: '<S700>/Signal Copy'
         *  Sum: '<S937>/Add' *)
        OP_ChiefMaster_Battery3_Msg13[0] := UDINT_TO_USINT(USINT_TO_UDINT(UDINT_TO_USINT(USINT_TO_UDINT(UDINT_TO_USINT(USINT_TO_UDINT(UDINT_TO_USINT(USINT_TO_UDINT(UDINT_TO_USINT(USINT_TO_UDINT(UDINT_TO_USINT(USINT_TO_UDINT(UDINT_TO_USINT(DINT_TO_UDINT(DWORD_TO_DINT(SHL(DINT_TO_DWORD(BOOL_TO_DINT(rtb_IP_boBMS_SDError_BB3)), 7))) + USINT_TO_UDINT(ShiftArithmetic5_f))) + USINT_TO_UDINT(BYTE_TO_USINT(SHL(USINT_TO_BYTE(DINT_TO_USINT(TRUNC(Count_k))), 5))))) + USINT_TO_UDINT(BYTE_TO_USINT(SHL(USINT_TO_BYTE(DINT_TO_USINT(TRUNC(y))), 4))))) + USINT_TO_UDINT(ShiftArithmetic2_h))) + USINT_TO_UDINT(BYTE_TO_USINT(SHL(USINT_TO_BYTE(DINT_TO_USINT(TRUNC(v))), 2))))) + OP_ChiefMaster_Battery3_Msg13_tmp)) + DINT_TO_UDINT(TRUNC(y_0)));
        (* Product: '<S948>/Divide' incorporates:
         *  Constant: '<S811>/Constant4'
         *  SignalConversion: '<S682>/BusConversion_InsertedFor_IT_BatterySignal_Databus_at_inport_0' *)
        rtb_Add_d := rtb_Add_j3 / 0.1;
        (* End of Outputs for SubSystem: '<S676>/BatteryPackSignals' *)
        

        (* DataTypeConversion: '<S944>/Data Type Conversion2' *)

        IF rtb_Add_d >= 0.5 THEN 
            rtb_Add_j3 := rt_floorf(u := rtb_Add_d + 0.5);
        ELSE 
            rtb_Add_j3 := 0.0;
        END_IF;

        (* Outputs for Atomic SubSystem: '<S676>/BatteryPackSignals' *)
        (* Product: '<S949>/Divide' incorporates:
         *  Constant: '<S811>/Constant3'
         *  SignalConversion: '<S682>/BusConversion_InsertedFor_IT_BatterySignal_Databus_at_inport_0' *)
        rtb_Add_d := rtb_Add_g / 0.1;
        (* End of Outputs for SubSystem: '<S676>/BatteryPackSignals' *)
        

        (* DataTypeConversion: '<S945>/Data Type Conversion2' *)

        IF rtb_Add_d >= 0.5 THEN 
            rtb_Add_g := rt_floorf(u := rtb_Add_d + 0.5);
        ELSE 
            rtb_Add_g := 0.0;
        END_IF;

        (* Outputs for Atomic SubSystem: '<S676>/BatteryPackSignals' *)
        (* Product: '<S950>/Divide' incorporates:
         *  Constant: '<S811>/Constant6'
         *  SignalConversion: '<S682>/BusConversion_InsertedFor_IT_BatterySignal_Databus_at_inport_0' *)
        rtb_Add_d := rtb_Add_ky / 100.0;
        (* End of Outputs for SubSystem: '<S676>/BatteryPackSignals' *)
        

        (* DataTypeConversion: '<S946>/Data Type Conversion2' *)
        rtb_Divide_h := ABS(rtb_Add_d);

        IF rtb_Divide_h < 8.388608E+6 THEN 

